  PROC DrawPart12()
    MoveL Offs(pOrigin,195.12,-45.16,-0.00),v40,z0,tcp\WObj:=Plywood;
    MoveL Offs(pOrigin,198.74,-44.14,-0.00),v40,z0,tcp\WObj:=Plywood;
    MoveL Offs(pOrigin,202.88,-41.55,-0.00),v40,z0,tcp\WObj:=Plywood;
    MoveL Offs(pOrigin,205.61,-38.96,-0.00),v40,z0,tcp\WObj:=Plywood;
    MoveL Offs(pOrigin,203.94,-41.12,-0.00),v40,z0,tcp\WObj:=Plywood;
    MoveL Offs(pOrigin,201.82,-42.93,-0.00),v40,z0,tcp\WObj:=Plywood;
    MoveL Offs(pOrigin,198.52,-44.77,-0.00),v40,z0,tcp\WObj:=Plywood;
    MoveL Offs(pOrigin,195.87,-45.59,-0.00),v40,z0,tcp\WObj:=Plywood;
    MoveL Offs(pOrigin,191.41,-45.80,-0.00),v40,z0,tcp\WObj:=Plywood;
    MoveL Offs(pOrigin,188.96,-45.38,-0.00),v40,z0,tcp\WObj:=Plywood;
    MoveL Offs(pOrigin,185.14,-44.24,-0.00),v40,z0,tcp\WObj:=Plywood;
    MoveL Offs(pOrigin,180.14,-41.51,-0.00),v40,z0,tcp\WObj:=Plywood;
    MoveL Offs(pOrigin,177.10,-41.34,-0.00),v40,z0,tcp\WObj:=Plywood;
    MoveL Offs(pOrigin,177.74,-41.62,-0.00),v40,z0,tcp\WObj:=Plywood;
    MoveL Offs(pOrigin,179.93,-44.53,-0.00),v40,z0,tcp\WObj:=Plywood;
    MoveL Offs(pOrigin,183.47,-47.75,-0.00),v40,z0,tcp\WObj:=Plywood;
    MoveL Offs(pOrigin,180.04,-45.06,-0.00),v40,z0,tcp\WObj:=Plywood;
    MoveL Offs(pOrigin,177.74,-41.62,-0.00),v40,fine,tcp\WObj:=Plywood;
    MoveL Offs(pOrigin,177.74,-41.62,-6.00),v60,z5,tcp\WObj:=Plywood;
    MoveL Offs(pOrigin,178.83,-45.34,-6.00),vTravel,z5,tcp\WObj:=Plywood;
    MoveL Offs(pOrigin,178.83,-45.34,-0.00),v60,z0,tcp\WObj:=Plywood;
    MoveL Offs(pOrigin,182.48,-49.09,-0.00),v40,z0,tcp\WObj:=Plywood;
    MoveL Offs(pOrigin,184.50,-50.30,-0.00),v40,z0,tcp\WObj:=Plywood;
    MoveL Offs(pOrigin,186.55,-51.01,-0.00),v40,z0,tcp\WObj:=Plywood;
    MoveL Offs(pOrigin,184.61,-50.51,-0.00),v40,z0,tcp\WObj:=Plywood;
    MoveL Offs(pOrigin,182.16,-49.20,-0.00),v40,z0,tcp\WObj:=Plywood;
    MoveL Offs(pOrigin,180.68,-47.92,-0.00),v40,z0,tcp\WObj:=Plywood;
    MoveL Offs(pOrigin,178.83,-45.34,-0.00),v40,fine,tcp\WObj:=Plywood;
    MoveL Offs(pOrigin,178.83,-45.34,-6.00),v60,z5,tcp\WObj:=Plywood;
    MoveL Offs(pOrigin,183.61,-42.29,-6.00),vTravel,z5,tcp\WObj:=Plywood;
    MoveL Offs(pOrigin,183.61,-42.29,-0.00),v60,z0,tcp\WObj:=Plywood;
    MoveL Offs(pOrigin,187.58,-42.61,-0.00),v40,z0,tcp\WObj:=Plywood;
    MoveL Offs(pOrigin,192.82,-41.76,-0.00),v40,z0,tcp\WObj:=Plywood;
    MoveL Offs(pOrigin,188.32,-42.83,-0.00),v40,z0,tcp\WObj:=Plywood;
    MoveL Offs(pOrigin,185.24,-42.72,-0.00),v40,z0,tcp\WObj:=Plywood;
    MoveL Offs(pOrigin,183.61,-42.29,-0.00),v40,fine,tcp\WObj:=Plywood;
    MoveL Offs(pOrigin,183.61,-42.29,-6.00),v60,z5,tcp\WObj:=Plywood;
    MoveL Offs(pOrigin,189.56,-46.22,-6.00),vTravel,z5,tcp\WObj:=Plywood;
    MoveL Offs(pOrigin,189.56,-46.22,-0.00),v60,z0,tcp\WObj:=Plywood;
    MoveL Offs(pOrigin,194.06,-47.29,-0.00),v40,z0,tcp\WObj:=Plywood;
    MoveL Offs(pOrigin,198.14,-47.08,-0.00),v40,z0,tcp\WObj:=Plywood;
    MoveL Offs(pOrigin,196.40,-47.50,-0.00),v40,z0,tcp\WObj:=Plywood;
    MoveL Offs(pOrigin,193.64,-47.50,-0.00),v40,z0,tcp\WObj:=Plywood;
    MoveL Offs(pOrigin,189.56,-46.22,-0.00),v40,fine,tcp\WObj:=Plywood;
    MoveL Offs(pOrigin,189.56,-46.22,-6.00),v60,z5,tcp\WObj:=Plywood;
    MoveL Offs(pOrigin,191.94,-54.30,-6.00),vTravel,z5,tcp\WObj:=Plywood;
    MoveL Offs(pOrigin,191.94,-54.30,-0.00),v60,z0,tcp\WObj:=Plywood;
    MoveL Offs(pOrigin,195.87,-53.17,-0.00),v40,z0,tcp\WObj:=Plywood;
    MoveL Offs(pOrigin,199.06,-51.68,-0.00),v40,z0,tcp\WObj:=Plywood;
    MoveL Offs(pOrigin,201.85,-49.70,-0.00),v40,z0,tcp\WObj:=Plywood;
    MoveL Offs(pOrigin,199.38,-51.79,-0.00),v40,z0,tcp\WObj:=Plywood;
    MoveL Offs(pOrigin,195.76,-53.59,-0.00),v40,z0,tcp\WObj:=Plywood;
    MoveL Offs(pOrigin,192.26,-54.62,-0.00),v40,z0,tcp\WObj:=Plywood;
    MoveL Offs(pOrigin,188.11,-55.15,-0.00),v40,z0,tcp\WObj:=Plywood;
    MoveL Offs(pOrigin,185.35,-54.94,-0.00),v40,z0,tcp\WObj:=Plywood;
    MoveL Offs(pOrigin,182.91,-54.23,-0.00),v40,z0,tcp\WObj:=Plywood;
    MoveL Offs(pOrigin,180.78,-52.71,-0.00),v40,z0,tcp\WObj:=Plywood;
    MoveL Offs(pOrigin,179.75,-51.01,-0.00),v40,z0,tcp\WObj:=Plywood;
    MoveL Offs(pOrigin,181.21,-52.81,-0.00),v40,z0,tcp\WObj:=Plywood;
    MoveL Offs(pOrigin,183.01,-53.91,-0.00),v40,z0,tcp\WObj:=Plywood;
    MoveL Offs(pOrigin,185.56,-54.62,-0.00),v40,z0,tcp\WObj:=Plywood;
    MoveL Offs(pOrigin,188.75,-54.72,-0.00),v40,z0,tcp\WObj:=Plywood;
    MoveL Offs(pOrigin,191.94,-54.30,-0.00),v40,fine,tcp\WObj:=Plywood;
    MoveL Offs(pOrigin,191.94,-54.30,-6.00),v60,z5,tcp\WObj:=Plywood;
    MoveL Offs(pOrigin,191.30,-56.64,-6.00),vTravel,z5,tcp\WObj:=Plywood;
    MoveL Offs(pOrigin,191.30,-56.64,-0.00),v60,z0,tcp\WObj:=Plywood;
    MoveL Offs(pOrigin,186.20,-56.96,-0.00),v40,z0,tcp\WObj:=Plywood;
    MoveL Offs(pOrigin,182.91,-56.42,-0.00),v40,z0,tcp\WObj:=Plywood;
    MoveL Offs(pOrigin,179.36,-55.04,-0.00),v40,z0,tcp\WObj:=Plywood;
    MoveL Offs(pOrigin,183.23,-56.32,-0.00),v40,z0,tcp\WObj:=Plywood;
    MoveL Offs(pOrigin,186.94,-56.74,-0.00),v40,z0,tcp\WObj:=Plywood;
    MoveL Offs(pOrigin,190.66,-56.53,-0.00),v40,z0,tcp\WObj:=Plywood;
    MoveL Offs(pOrigin,195.59,-55.36,-0.00),v40,z0,tcp\WObj:=Plywood;
    MoveL Offs(pOrigin,191.30,-56.64,-0.00),v40,fine,tcp\WObj:=Plywood;
    MoveL Offs(pOrigin,191.30,-56.64,-6.00),v60,z5,tcp\WObj:=Plywood;
    MoveL Offs(pOrigin,195.80,-66.84,-6.00),vTravel,z5,tcp\WObj:=Plywood;
    MoveL Offs(pOrigin,195.80,-66.84,-0.00),v60,z0,tcp\WObj:=Plywood;
    MoveL Offs(pOrigin,195.44,-67.69,-0.00),v40,z0,tcp\WObj:=Plywood;
    MoveL Offs(pOrigin,195.23,-71.94,-0.00),v40,z0,tcp\WObj:=Plywood;
    MoveL Offs(pOrigin,194.70,-73.21,-0.00),v40,z0,tcp\WObj:=Plywood;
    MoveL Offs(pOrigin,193.39,-74.70,-0.00),v40,z0,tcp\WObj:=Plywood;
    MoveL Offs(pOrigin,193.43,-77.57,-0.00),v40,z0,tcp\WObj:=Plywood;
    MoveL Offs(pOrigin,191.16,-82.56,-0.00),v40,z0,tcp\WObj:=Plywood;
    MoveL Offs(pOrigin,190.34,-85.22,-0.00),v40,z0,tcp\WObj:=Plywood;
    MoveL Offs(pOrigin,190.88,-87.88,-0.00),v40,z0,tcp\WObj:=Plywood;
    MoveL Offs(pOrigin,189.18,-94.25,-0.00),v40,z0,tcp\WObj:=Plywood;
    MoveL Offs(pOrigin,190.66,-103.81,-0.00),v40,z0,tcp\WObj:=Plywood;
    MoveL Offs(pOrigin,190.88,-111.68,-0.00),v40,z0,tcp\WObj:=Plywood;
    MoveL Offs(pOrigin,190.13,-116.56,-0.00),v40,z0,tcp\WObj:=Plywood;
    MoveL Offs(pOrigin,188.86,-119.68,-0.00),v40,z0,tcp\WObj:=Plywood;
    MoveL Offs(pOrigin,190.80,-116.88,-0.00),v40,z0,tcp\WObj:=Plywood;
    MoveL Offs(pOrigin,192.15,-111.57,-0.00),v40,z0,tcp\WObj:=Plywood;
    MoveL Offs(pOrigin,196.40,-67.47,-0.00),v40,z0,tcp\WObj:=Plywood;
    MoveL Offs(pOrigin,196.19,-66.73,-0.00),v40,z0,tcp\WObj:=Plywood;
    MoveL Offs(pOrigin,195.80,-66.84,-0.00),v40,fine,tcp\WObj:=Plywood;
    MoveL Offs(pOrigin,195.80,-66.84,-6.00),v60,z5,tcp\WObj:=Plywood;
    MoveL Offs(pOrigin,193.35,-71.19,-6.00),vTravel,z5,tcp\WObj:=Plywood;
    MoveL Offs(pOrigin,193.35,-71.19,-0.00),v60,z0,tcp\WObj:=Plywood;
    MoveL Offs(pOrigin,191.19,-71.09,-0.00),v40,z0,tcp\WObj:=Plywood;
    MoveL Offs(pOrigin,188.18,-69.64,-0.00),v40,z0,tcp\WObj:=Plywood;
    MoveL Offs(pOrigin,191.30,-70.88,-0.00),v40,z0,tcp\WObj:=Plywood;
    MoveL Offs(pOrigin,193.35,-71.19,-0.00),v40,fine,tcp\WObj:=Plywood;
    MoveL Offs(pOrigin,193.35,-71.19,-6.00),v60,z5,tcp\WObj:=Plywood;
    MoveL Offs(pOrigin,181.52,-78.17,-6.00),vTravel,z5,tcp\WObj:=Plywood;
    MoveL Offs(pOrigin,181.52,-78.17,-0.00),v60,z0,tcp\WObj:=Plywood;
    MoveL Offs(pOrigin,188.04,-89.11,-0.00),v40,z0,tcp\WObj:=Plywood;
    MoveL Offs(pOrigin,184.68,-84.16,-0.00),v40,z0,tcp\WObj:=Plywood;
    MoveL Offs(pOrigin,181.52,-78.17,-0.00),v40,fine,tcp\WObj:=Plywood;
    MoveL Offs(pOrigin,181.52,-78.17,-6.00),v60,z5,tcp\WObj:=Plywood;
    MoveL Offs(pOrigin,172.25,-67.05,-6.00),vTravel,z5,tcp\WObj:=Plywood;
    MoveL Offs(pOrigin,172.25,-67.05,-0.00),v60,z0,tcp\WObj:=Plywood;
    MoveL Offs(pOrigin,172.49,-63.33,-0.00),v40,z0,tcp\WObj:=Plywood;
    MoveL Offs(pOrigin,172.18,-61.88,-0.00),v40,z0,tcp\WObj:=Plywood;
    MoveL Offs(pOrigin,152.73,-56.53,-0.00),v40,z0,tcp\WObj:=Plywood;
    MoveL Offs(pOrigin,148.16,-55.47,-0.00),v40,z0,tcp\WObj:=Plywood;
    MoveL Offs(pOrigin,147.49,-55.79,-0.00),v40,z0,tcp\WObj:=Plywood;
    MoveL Offs(pOrigin,149.01,-60.60,-0.00),v40,z0,tcp\WObj:=Plywood;
    MoveL Offs(pOrigin,172.25,-67.05,-0.00),v40,fine,tcp\WObj:=Plywood;
    MoveL Offs(pOrigin,172.25,-67.05,-6.00),v60,z5,tcp\WObj:=Plywood;
    MoveL Offs(pOrigin,170.83,-65.56,-6.00),vTravel,z5,tcp\WObj:=Plywood;
  ENDPROC

  PROC DrawPart13()
    MoveL Offs(pOrigin,170.83,-65.56,-0.00),v60,z0,tcp\WObj:=Plywood;
    MoveL Offs(pOrigin,151.00,-60.14,-0.00),v40,z0,tcp\WObj:=Plywood;
    MoveL Offs(pOrigin,170.83,-65.56,-0.00),v40,fine,tcp\WObj:=Plywood;
    MoveL Offs(pOrigin,170.83,-65.56,-6.00),v60,z5,tcp\WObj:=Plywood;
    MoveL Offs(pOrigin,155.00,-73.39,-6.00),vTravel,z5,tcp\WObj:=Plywood;
    MoveL Offs(pOrigin,155.00,-73.39,-0.00),v60,z0,tcp\WObj:=Plywood;
    MoveL Offs(pOrigin,158.43,-79.38,-0.00),v40,z0,tcp\WObj:=Plywood;
    MoveL Offs(pOrigin,162.08,-84.58,-0.00),v40,z0,tcp\WObj:=Plywood;
    MoveL Offs(pOrigin,165.48,-88.62,-0.00),v40,z0,tcp\WObj:=Plywood;
    MoveL Offs(pOrigin,170.09,-92.90,-0.00),v40,z0,tcp\WObj:=Plywood;
    MoveL Offs(pOrigin,167.07,-90.53,-0.00),v40,z0,tcp\WObj:=Plywood;
    MoveL Offs(pOrigin,161.76,-84.69,-0.00),v40,z0,tcp\WObj:=Plywood;
    MoveL Offs(pOrigin,157.90,-78.95,-0.00),v40,z0,tcp\WObj:=Plywood;
    MoveL Offs(pOrigin,155.00,-73.39,-0.00),v40,fine,tcp\WObj:=Plywood;
    MoveL Offs(pOrigin,155.00,-73.39,-6.00),v60,z5,tcp\WObj:=Plywood;
    MoveL Offs(pOrigin,152.62,-86.92,-6.00),vTravel,z5,tcp\WObj:=Plywood;
    MoveL Offs(pOrigin,152.62,-86.92,-0.00),v60,z0,tcp\WObj:=Plywood;
    MoveL Offs(pOrigin,153.12,-87.13,-0.00),v40,z0,tcp\WObj:=Plywood;
    MoveL Offs(pOrigin,153.05,-87.52,-0.00),v40,z0,tcp\WObj:=Plywood;
    MoveL Offs(pOrigin,148.27,-89.26,-0.00),v40,z0,tcp\WObj:=Plywood;
    MoveL Offs(pOrigin,147.63,-89.15,-0.00),v40,z0,tcp\WObj:=Plywood;
    MoveL Offs(pOrigin,151.35,-87.31,-0.00),v40,z0,tcp\WObj:=Plywood;
    MoveL Offs(pOrigin,152.62,-86.92,-0.00),v40,z0,tcp\WObj:=Plywood;
    MoveL Offs(pOrigin,152.84,-87.24,-0.00),v40,z0,tcp\WObj:=Plywood;
    MoveL Offs(pOrigin,151.14,-87.63,-0.00),v40,z0,tcp\WObj:=Plywood;
    MoveL Offs(pOrigin,148.55,-88.83,-0.00),v40,z0,tcp\WObj:=Plywood;
    MoveL Offs(pOrigin,151.14,-88.12,-0.00),v40,z0,tcp\WObj:=Plywood;
    MoveL Offs(pOrigin,152.84,-87.24,-0.00),v40,fine,tcp\WObj:=Plywood;
    MoveL Offs(pOrigin,152.84,-87.24,-6.00),v60,z5,tcp\WObj:=Plywood;
    MoveL Offs(pOrigin,159.32,-88.58,-6.00),vTravel,z5,tcp\WObj:=Plywood;
    MoveL Offs(pOrigin,159.32,-88.58,-0.00),v60,z0,tcp\WObj:=Plywood;
    MoveL Offs(pOrigin,160.38,-92.02,-0.00),v40,z0,tcp\WObj:=Plywood;
    MoveL Offs(pOrigin,160.49,-94.89,-0.00),v40,z0,tcp\WObj:=Plywood;
    MoveL Offs(pOrigin,159.50,-98.18,-0.00),v40,z0,tcp\WObj:=Plywood;
    MoveL Offs(pOrigin,157.65,-100.87,-0.00),v40,z0,tcp\WObj:=Plywood;
    MoveL Offs(pOrigin,159.25,-98.18,-0.00),v40,z0,tcp\WObj:=Plywood;
    MoveL Offs(pOrigin,160.17,-95.10,-0.00),v40,z0,tcp\WObj:=Plywood;
    MoveL Offs(pOrigin,160.17,-92.12,-0.00),v40,z0,tcp\WObj:=Plywood;
    MoveL Offs(pOrigin,159.32,-88.58,-0.00),v40,fine,tcp\WObj:=Plywood;
    MoveL Offs(pOrigin,159.32,-88.58,-6.00),v60,z5,tcp\WObj:=Plywood;
    MoveL Offs(pOrigin,156.98,-99.92,-6.00),vTravel,z5,tcp\WObj:=Plywood;
    MoveL Offs(pOrigin,156.98,-99.92,-0.00),v60,z0,tcp\WObj:=Plywood;
    MoveL Offs(pOrigin,150.71,-97.01,-0.00),v40,z0,tcp\WObj:=Plywood;
    MoveL Offs(pOrigin,143.81,-102.01,-0.00),v40,z0,tcp\WObj:=Plywood;
    MoveL Offs(pOrigin,144.87,-109.02,-0.00),v40,z0,tcp\WObj:=Plywood;
    MoveL Offs(pOrigin,144.59,-114.54,-0.00),v40,z0,tcp\WObj:=Plywood;
    MoveL Offs(pOrigin,151.24,-107.43,-0.00),v40,z0,tcp\WObj:=Plywood;
    MoveL Offs(pOrigin,156.98,-99.92,-0.00),v40,fine,tcp\WObj:=Plywood;
    MoveL Offs(pOrigin,156.98,-99.92,-6.00),v60,z5,tcp\WObj:=Plywood;
    MoveL Offs(pOrigin,158.36,-107.04,-6.00),vTravel,z5,tcp\WObj:=Plywood;
    MoveL Offs(pOrigin,158.36,-107.04,-0.00),v60,z0,tcp\WObj:=Plywood;
    MoveL Offs(pOrigin,150.50,-109.30,-0.00),v40,z0,tcp\WObj:=Plywood;
    MoveL Offs(pOrigin,147.10,-112.63,-0.00),v40,z0,tcp\WObj:=Plywood;
    MoveL Offs(pOrigin,144.59,-115.71,-0.00),v40,z0,tcp\WObj:=Plywood;
    MoveL Offs(pOrigin,145.51,-118.47,-0.00),v40,z0,tcp\WObj:=Plywood;
    MoveL Offs(pOrigin,145.97,-121.34,-0.00),v40,z0,tcp\WObj:=Plywood;
    MoveL Offs(pOrigin,147.31,-121.34,-0.00),v40,z0,tcp\WObj:=Plywood;
    MoveL Offs(pOrigin,148.69,-122.19,-0.00),v40,z0,tcp\WObj:=Plywood;
    MoveL Offs(pOrigin,162.61,-121.88,-0.00),v40,z0,tcp\WObj:=Plywood;
    MoveL Offs(pOrigin,175.79,-120.60,-0.00),v40,z0,tcp\WObj:=Plywood;
    MoveL Offs(pOrigin,181.21,-119.54,-0.00),v40,z0,tcp\WObj:=Plywood;
    MoveL Offs(pOrigin,183.23,-118.72,-0.00),v40,z0,tcp\WObj:=Plywood;
    MoveL Offs(pOrigin,184.50,-117.84,-0.00),v40,z0,tcp\WObj:=Plywood;
    MoveL Offs(pOrigin,186.02,-116.03,-0.00),v40,z0,tcp\WObj:=Plywood;
    MoveL Offs(pOrigin,187.26,-112.95,-0.00),v40,z0,tcp\WObj:=Plywood;
    MoveL Offs(pOrigin,187.79,-110.08,-0.00),v40,z0,tcp\WObj:=Plywood;
    MoveL Offs(pOrigin,187.79,-105.62,-0.00),v40,z0,tcp\WObj:=Plywood;
    MoveL Offs(pOrigin,186.27,-97.97,-0.00),v40,z0,tcp\WObj:=Plywood;
    MoveL Offs(pOrigin,185.77,-97.76,-0.00),v40,z0,tcp\WObj:=Plywood;
    MoveL Offs(pOrigin,171.64,-101.79,-0.00),v40,z0,tcp\WObj:=Plywood;
    MoveL Offs(pOrigin,158.36,-107.04,-0.00),v40,fine,tcp\WObj:=Plywood;
    MoveL Offs(pOrigin,158.36,-107.04,-6.00),v60,z5,tcp\WObj:=Plywood;
    MoveL Offs(pOrigin,156.02,-122.62,-6.00),vTravel,z5,tcp\WObj:=Plywood;
    MoveL Offs(pOrigin,156.02,-122.62,-0.00),v60,z0,tcp\WObj:=Plywood;
    MoveL Offs(pOrigin,149.01,-122.44,-0.00),v40,z0,tcp\WObj:=Plywood;
    MoveL Offs(pOrigin,149.54,-124.96,-0.00),v40,z0,tcp\WObj:=Plywood;
    MoveL Offs(pOrigin,158.26,-125.06,-0.00),v40,z0,tcp\WObj:=Plywood;
    MoveL Offs(pOrigin,172.28,-124.21,-0.00),v40,z0,tcp\WObj:=Plywood;
    MoveL Offs(pOrigin,181.95,-122.94,-0.00),v40,z0,tcp\WObj:=Plywood;
    MoveL Offs(pOrigin,185.03,-122.12,-0.00),v40,z0,tcp\WObj:=Plywood;
    MoveL Offs(pOrigin,186.94,-121.24,-0.00),v40,z0,tcp\WObj:=Plywood;
    MoveL Offs(pOrigin,188.57,-119.22,-0.00),v40,z0,tcp\WObj:=Plywood;
    MoveL Offs(pOrigin,189.32,-117.52,-0.00),v40,z0,tcp\WObj:=Plywood;
    MoveL Offs(pOrigin,190.24,-112.31,-0.00),v40,z0,tcp\WObj:=Plywood;
    MoveL Offs(pOrigin,190.24,-105.83,-0.00),v40,z0,tcp\WObj:=Plywood;
    MoveL Offs(pOrigin,189.07,-95.31,-0.00),v40,z0,tcp\WObj:=Plywood;
    MoveL Offs(pOrigin,188.22,-96.59,-0.00),v40,z0,tcp\WObj:=Plywood;
    MoveL Offs(pOrigin,186.84,-97.76,-0.00),v40,z0,tcp\WObj:=Plywood;
    MoveL Offs(pOrigin,188.64,-106.89,-0.00),v40,z0,tcp\WObj:=Plywood;
    MoveL Offs(pOrigin,188.86,-109.97,-0.00),v40,z0,tcp\WObj:=Plywood;
    MoveL Offs(pOrigin,188.64,-114.86,-0.00),v40,z0,tcp\WObj:=Plywood;
    MoveL Offs(pOrigin,187.51,-118.69,-0.00),v40,z0,tcp\WObj:=Plywood;
    MoveL Offs(pOrigin,185.67,-120.81,-0.00),v40,z0,tcp\WObj:=Plywood;
    MoveL Offs(pOrigin,182.59,-122.09,-0.00),v40,z0,tcp\WObj:=Plywood;
    MoveL Offs(pOrigin,179.15,-122.26,-0.00),v40,z0,tcp\WObj:=Plywood;
    MoveL Offs(pOrigin,183.86,-121.06,-0.00),v40,z0,tcp\WObj:=Plywood;
    MoveL Offs(pOrigin,185.24,-120.28,-0.00),v40,z0,tcp\WObj:=Plywood;
    MoveL Offs(pOrigin,186.41,-119.11,-0.00),v40,z0,tcp\WObj:=Plywood;
    MoveL Offs(pOrigin,187.30,-117.52,-0.00),v40,z0,tcp\WObj:=Plywood;
    MoveL Offs(pOrigin,188.01,-114.86,-0.00),v40,z0,tcp\WObj:=Plywood;
    MoveL Offs(pOrigin,188.22,-112.84,-0.00),v40,z0,tcp\WObj:=Plywood;
    MoveL Offs(pOrigin,188.01,-109.41,-0.00),v40,z0,tcp\WObj:=Plywood;
    MoveL Offs(pOrigin,187.48,-112.84,-0.00),v40,z0,tcp\WObj:=Plywood;
    MoveL Offs(pOrigin,186.13,-116.24,-0.00),v40,z0,tcp\WObj:=Plywood;
    MoveL Offs(pOrigin,184.39,-118.26,-0.00),v40,z0,tcp\WObj:=Plywood;
    MoveL Offs(pOrigin,182.38,-119.47,-0.00),v40,z0,tcp\WObj:=Plywood;
    MoveL Offs(pOrigin,177.81,-120.71,-0.00),v40,z0,tcp\WObj:=Plywood;
    MoveL Offs(pOrigin,168.67,-121.88,-0.00),v40,z0,tcp\WObj:=Plywood;
    MoveL Offs(pOrigin,156.02,-122.62,-0.00),v40,fine,tcp\WObj:=Plywood;
    MoveL Offs(pOrigin,156.02,-122.62,-6.00),v60,z5,tcp\WObj:=Plywood;
    MoveL Offs(pOrigin,148.41,-123.04,-6.00),vTravel,z5,tcp\WObj:=Plywood;
    MoveL Offs(pOrigin,148.41,-123.04,-0.00),v60,z0,tcp\WObj:=Plywood;
    MoveL Offs(pOrigin,147.52,-122.02,-0.00),v40,z0,tcp\WObj:=Plywood;
    MoveL Offs(pOrigin,146.78,-121.88,-0.00),v40,z0,tcp\WObj:=Plywood;
    MoveL Offs(pOrigin,146.14,-122.19,-0.00),v40,z0,tcp\WObj:=Plywood;
    MoveL Offs(pOrigin,145.29,-126.27,-0.00),v40,z0,tcp\WObj:=Plywood;
    MoveL Offs(pOrigin,145.51,-122.72,-0.00),v40,z0,tcp\WObj:=Plywood;
    MoveL Offs(pOrigin,144.76,-118.05,-0.00),v40,z0,tcp\WObj:=Plywood;
    MoveL Offs(pOrigin,143.31,-114.76,-0.00),v40,z0,tcp\WObj:=Plywood;
    MoveL Offs(pOrigin,140.23,-110.15,-0.00),v40,z0,tcp\WObj:=Plywood;
  ENDPROC

  PROC DrawPart14()
    MoveL Offs(pOrigin,143.59,-114.37,-0.00),v40,z0,tcp\WObj:=Plywood;
    MoveL Offs(pOrigin,142.35,-110.40,-0.00),v40,z0,tcp\WObj:=Plywood;
    MoveL Offs(pOrigin,141.08,-107.85,-0.00),v40,z0,tcp\WObj:=Plywood;
    MoveL Offs(pOrigin,139.56,-105.83,-0.00),v40,z0,tcp\WObj:=Plywood;
    MoveL Offs(pOrigin,134.85,-102.15,-0.00),v40,z0,tcp\WObj:=Plywood;
    MoveL Offs(pOrigin,137.75,-103.81,-0.00),v40,z0,tcp\WObj:=Plywood;
    MoveL Offs(pOrigin,139.84,-105.51,-0.00),v40,z0,tcp\WObj:=Plywood;
    MoveL Offs(pOrigin,137.96,-102.22,-0.00),v40,z0,tcp\WObj:=Plywood;
    MoveL Offs(pOrigin,135.52,-100.27,-0.00),v40,z0,tcp\WObj:=Plywood;
    MoveL Offs(pOrigin,132.86,-98.89,-0.00),v40,z0,tcp\WObj:=Plywood;
    MoveL Offs(pOrigin,129.89,-98.07,-0.00),v40,z0,tcp\WObj:=Plywood;
    MoveL Offs(pOrigin,126.66,-98.39,-0.00),v40,z0,tcp\WObj:=Plywood;
    MoveL Offs(pOrigin,128.93,-97.86,-0.00),v40,z0,tcp\WObj:=Plywood;
    MoveL Offs(pOrigin,131.38,-98.18,-0.00),v40,z0,tcp\WObj:=Plywood;
    MoveL Offs(pOrigin,133.39,-98.89,-0.00),v40,z0,tcp\WObj:=Plywood;
    MoveL Offs(pOrigin,137.40,-101.16,-0.00),v40,z0,tcp\WObj:=Plywood;
    MoveL Offs(pOrigin,135.52,-98.18,-0.00),v40,z0,tcp\WObj:=Plywood;
    MoveL Offs(pOrigin,134.46,-97.12,-0.00),v40,z0,tcp\WObj:=Plywood;
    MoveL Offs(pOrigin,130.81,-95.21,-0.00),v40,z0,tcp\WObj:=Plywood;
    MoveL Offs(pOrigin,134.53,-96.69,-0.00),v40,z0,tcp\WObj:=Plywood;
    MoveL Offs(pOrigin,130.84,-91.70,-0.00),v40,z0,tcp\WObj:=Plywood;
    MoveL Offs(pOrigin,129.04,-86.92,-0.00),v40,z0,tcp\WObj:=Plywood;
    MoveL Offs(pOrigin,126.49,-84.72,-0.00),v40,z0,tcp\WObj:=Plywood;
    MoveL Offs(pOrigin,122.73,-87.98,-0.00),v40,z0,tcp\WObj:=Plywood;
    MoveL Offs(pOrigin,121.00,-92.76,-0.00),v40,z0,tcp\WObj:=Plywood;
    MoveL Offs(pOrigin,122.59,-92.27,-0.00),v40,z0,tcp\WObj:=Plywood;
    MoveL Offs(pOrigin,120.64,-93.40,-0.00),v40,z0,tcp\WObj:=Plywood;
    MoveL Offs(pOrigin,119.40,-95.63,-0.00),v40,z0,tcp\WObj:=Plywood;
    MoveL Offs(pOrigin,123.44,-94.46,-0.00),v40,z0,tcp\WObj:=Plywood;
    MoveL Offs(pOrigin,121.18,-95.17,-0.00),v40,z0,tcp\WObj:=Plywood;
    MoveL Offs(pOrigin,118.62,-96.69,-0.00),v40,z0,tcp\WObj:=Plywood;
    MoveL Offs(pOrigin,116.22,-100.09,-0.00),v40,z0,tcp\WObj:=Plywood;
    MoveL Offs(pOrigin,119.16,-98.57,-0.00),v40,z0,tcp\WObj:=Plywood;
    MoveL Offs(pOrigin,122.27,-97.97,-0.00),v40,z0,tcp\WObj:=Plywood;
    MoveL Offs(pOrigin,119.16,-98.78,-0.00),v40,z0,tcp\WObj:=Plywood;
    MoveL Offs(pOrigin,116.29,-100.62,-0.00),v40,z0,tcp\WObj:=Plywood;
    MoveL Offs(pOrigin,114.80,-102.32,-0.00),v40,z0,tcp\WObj:=Plywood;
    MoveL Offs(pOrigin,113.95,-103.99,-0.00),v40,z0,tcp\WObj:=Plywood;
    MoveL Offs(pOrigin,116.93,-102.29,-0.00),v40,z0,tcp\WObj:=Plywood;
    MoveL Offs(pOrigin,119.62,-101.37,-0.00),v40,z0,tcp\WObj:=Plywood;
    MoveL Offs(pOrigin,116.50,-102.82,-0.00),v40,z0,tcp\WObj:=Plywood;
    MoveL Offs(pOrigin,113.84,-104.66,-0.00),v40,z0,tcp\WObj:=Plywood;
    MoveL Offs(pOrigin,110.37,-108.28,-0.00),v40,z0,tcp\WObj:=Plywood;
    MoveL Offs(pOrigin,113.24,-107.11,-0.00),v40,z0,tcp\WObj:=Plywood;
    MoveL Offs(pOrigin,110.02,-108.91,-0.00),v40,z0,tcp\WObj:=Plywood;
    MoveL Offs(pOrigin,107.04,-111.68,-0.00),v40,z0,tcp\WObj:=Plywood;
    MoveL Offs(pOrigin,104.99,-115.18,-0.00),v40,z0,tcp\WObj:=Plywood;
    MoveL Offs(pOrigin,103.54,-121.06,-0.00),v40,z0,tcp\WObj:=Plywood;
    MoveL Offs(pOrigin,103.82,-116.67,-0.00),v40,z0,tcp\WObj:=Plywood;
    MoveL Offs(pOrigin,103.01,-116.70,-0.00),v40,z0,tcp\WObj:=Plywood;
    MoveL Offs(pOrigin,102.19,-117.52,-0.00),v40,z0,tcp\WObj:=Plywood;
    MoveL Offs(pOrigin,100.92,-123.68,-0.00),v40,z0,tcp\WObj:=Plywood;
    MoveL Offs(pOrigin,98.12,-129.42,-0.00),v40,z0,tcp\WObj:=Plywood;
    MoveL Offs(pOrigin,98.01,-130.91,-0.00),v40,z0,tcp\WObj:=Plywood;
    MoveL Offs(pOrigin,98.40,-132.93,-0.00),v40,z0,tcp\WObj:=Plywood;
    MoveL Offs(pOrigin,98.97,-133.77,-0.00),v40,z0,tcp\WObj:=Plywood;
    MoveL Offs(pOrigin,100.14,-134.20,-0.00),v40,z0,tcp\WObj:=Plywood;
    MoveL Offs(pOrigin,101.20,-133.56,-0.00),v40,z0,tcp\WObj:=Plywood;
    MoveL Offs(pOrigin,101.70,-132.61,-0.00),v40,z0,tcp\WObj:=Plywood;
    MoveL Offs(pOrigin,101.62,-132.04,-0.00),v40,z0,tcp\WObj:=Plywood;
    MoveL Offs(pOrigin,100.03,-132.71,-0.00),v40,z0,tcp\WObj:=Plywood;
    MoveL Offs(pOrigin,99.39,-132.61,-0.00),v40,z0,tcp\WObj:=Plywood;
    MoveL Offs(pOrigin,98.97,-130.16,-0.00),v40,z0,tcp\WObj:=Plywood;
    MoveL Offs(pOrigin,99.96,-127.68,-0.00),v40,z0,tcp\WObj:=Plywood;
    MoveL Offs(pOrigin,99.18,-129.84,-0.00),v40,z0,tcp\WObj:=Plywood;
    MoveL Offs(pOrigin,99.46,-131.86,-0.00),v40,z0,tcp\WObj:=Plywood;
    MoveL Offs(pOrigin,100.35,-132.29,-0.00),v40,z0,tcp\WObj:=Plywood;
    MoveL Offs(pOrigin,101.59,-131.23,-0.00),v40,z0,tcp\WObj:=Plywood;
    MoveL Offs(pOrigin,102.72,-127.08,-0.00),v40,z0,tcp\WObj:=Plywood;
    MoveL Offs(pOrigin,103.22,-126.55,-0.00),v40,z0,tcp\WObj:=Plywood;
    MoveL Offs(pOrigin,103.18,-124.00,-0.00),v40,z0,tcp\WObj:=Plywood;
    MoveL Offs(pOrigin,102.58,-124.85,-0.00),v40,z0,tcp\WObj:=Plywood;
    MoveL Offs(pOrigin,102.55,-126.48,-0.00),v40,z0,tcp\WObj:=Plywood;
    MoveL Offs(pOrigin,102.37,-124.64,-0.00),v40,z0,tcp\WObj:=Plywood;
    MoveL Offs(pOrigin,103.40,-122.55,-0.00),v40,z0,tcp\WObj:=Plywood;
    MoveL Offs(pOrigin,103.54,-131.90,-0.00),v40,z0,tcp\WObj:=Plywood;
    MoveL Offs(pOrigin,104.64,-128.99,-0.00),v40,z0,tcp\WObj:=Plywood;
    MoveL Offs(pOrigin,105.24,-128.04,-0.00),v40,z0,tcp\WObj:=Plywood;
    MoveL Offs(pOrigin,106.09,-127.47,-0.00),v40,z0,tcp\WObj:=Plywood;
    MoveL Offs(pOrigin,109.38,-127.08,-0.00),v40,z0,tcp\WObj:=Plywood;
    MoveL Offs(pOrigin,114.06,-127.61,-0.00),v40,z0,tcp\WObj:=Plywood;
    MoveL Offs(pOrigin,116.18,-128.21,-0.00),v40,z0,tcp\WObj:=Plywood;
    MoveL Offs(pOrigin,117.56,-129.21,-0.00),v40,z0,tcp\WObj:=Plywood;
    MoveL Offs(pOrigin,118.84,-131.01,-0.00),v40,z0,tcp\WObj:=Plywood;
    MoveL Offs(pOrigin,119.16,-134.41,-0.00),v40,z0,tcp\WObj:=Plywood;
    MoveL Offs(pOrigin,118.73,-134.09,-0.00),v40,z0,tcp\WObj:=Plywood;
    MoveL Offs(pOrigin,118.80,-134.73,-0.00),v40,z0,tcp\WObj:=Plywood;
    MoveL Offs(pOrigin,119.37,-135.19,-0.00),v40,z0,tcp\WObj:=Plywood;
    MoveL Offs(pOrigin,121.18,-135.58,-0.00),v40,z0,tcp\WObj:=Plywood;
    MoveL Offs(pOrigin,122.45,-135.26,-0.00),v40,z0,tcp\WObj:=Plywood;
    MoveL Offs(pOrigin,123.16,-132.71,-0.00),v40,z0,tcp\WObj:=Plywood;
    MoveL Offs(pOrigin,125.85,-129.81,-0.00),v40,z0,tcp\WObj:=Plywood;
    MoveL Offs(pOrigin,127.34,-129.42,-0.00),v40,z0,tcp\WObj:=Plywood;
    MoveL Offs(pOrigin,132.01,-129.63,-0.00),v40,z0,tcp\WObj:=Plywood;
    MoveL Offs(pOrigin,135.41,-130.38,-0.00),v40,z0,tcp\WObj:=Plywood;
    MoveL Offs(pOrigin,137.54,-131.44,-0.00),v40,z0,tcp\WObj:=Plywood;
    MoveL Offs(pOrigin,138.28,-133.46,-0.00),v40,z0,tcp\WObj:=Plywood;
    MoveL Offs(pOrigin,138.53,-137.28,-0.00),v40,z0,tcp\WObj:=Plywood;
    MoveL Offs(pOrigin,140.73,-137.88,-0.00),v40,z0,tcp\WObj:=Plywood;
    MoveL Offs(pOrigin,141.57,-137.88,-0.00),v40,z0,tcp\WObj:=Plywood;
    MoveL Offs(pOrigin,141.96,-137.39,-0.00),v40,z0,tcp\WObj:=Plywood;
    MoveL Offs(pOrigin,143.35,-132.61,-0.00),v40,z0,tcp\WObj:=Plywood;
    MoveL Offs(pOrigin,143.88,-131.76,-0.00),v40,z0,tcp\WObj:=Plywood;
    MoveL Offs(pOrigin,144.55,-132.89,-0.00),v40,z0,tcp\WObj:=Plywood;
    MoveL Offs(pOrigin,145.86,-130.91,-0.00),v40,z0,tcp\WObj:=Plywood;
    MoveL Offs(pOrigin,146.04,-129.74,-0.00),v40,z0,tcp\WObj:=Plywood;
    MoveL Offs(pOrigin,145.19,-127.61,-0.00),v40,z0,tcp\WObj:=Plywood;
    MoveL Offs(pOrigin,145.40,-127.15,-0.00),v40,z0,tcp\WObj:=Plywood;
    MoveL Offs(pOrigin,147.14,-129.21,-0.00),v40,z0,tcp\WObj:=Plywood;
    MoveL Offs(pOrigin,147.42,-130.62,-0.00),v40,z0,tcp\WObj:=Plywood;
    MoveL Offs(pOrigin,146.78,-129.31,-0.00),v40,z0,tcp\WObj:=Plywood;
    MoveL Offs(pOrigin,146.18,-128.89,-0.00),v40,z0,tcp\WObj:=Plywood;
    MoveL Offs(pOrigin,146.46,-130.27,-0.00),v40,z0,tcp\WObj:=Plywood;
    MoveL Offs(pOrigin,145.08,-132.71,-0.00),v40,z0,tcp\WObj:=Plywood;
    MoveL Offs(pOrigin,145.19,-133.14,-0.00),v40,z0,tcp\WObj:=Plywood;
    MoveL Offs(pOrigin,145.86,-133.17,-0.00),v40,z0,tcp\WObj:=Plywood;
    MoveL Offs(pOrigin,145.19,-133.56,-0.00),v40,z0,tcp\WObj:=Plywood;
    MoveL Offs(pOrigin,145.08,-133.99,-0.00),v40,z0,tcp\WObj:=Plywood;
    MoveL Offs(pOrigin,146.36,-136.64,-0.00),v40,z0,tcp\WObj:=Plywood;
    MoveL Offs(pOrigin,147.52,-137.74,-0.00),v40,z0,tcp\WObj:=Plywood;
  ENDPROC

  PROC DrawPart15()
    MoveL Offs(pOrigin,148.27,-137.92,-0.00),v40,z0,tcp\WObj:=Plywood;
    MoveL Offs(pOrigin,149.47,-136.64,-0.00),v40,z0,tcp\WObj:=Plywood;
    MoveL Offs(pOrigin,149.86,-133.99,-0.00),v40,z0,tcp\WObj:=Plywood;
    MoveL Offs(pOrigin,149.23,-131.90,-0.00),v40,z0,tcp\WObj:=Plywood;
    MoveL Offs(pOrigin,148.27,-135.19,-0.00),v40,z0,tcp\WObj:=Plywood;
    MoveL Offs(pOrigin,149.01,-131.12,-0.00),v40,z0,tcp\WObj:=Plywood;
    MoveL Offs(pOrigin,148.52,-128.99,-0.00),v40,z0,tcp\WObj:=Plywood;
    MoveL Offs(pOrigin,147.67,-127.36,-0.00),v40,z0,tcp\WObj:=Plywood;
    MoveL Offs(pOrigin,148.73,-128.99,-0.00),v40,z0,tcp\WObj:=Plywood;
    MoveL Offs(pOrigin,149.97,-133.88,-0.00),v40,z0,tcp\WObj:=Plywood;
    MoveL Offs(pOrigin,150.07,-135.05,-0.00),v40,z0,tcp\WObj:=Plywood;
    MoveL Offs(pOrigin,149.69,-136.75,-0.00),v40,z0,tcp\WObj:=Plywood;
    MoveL Offs(pOrigin,148.59,-138.17,-0.00),v40,z0,tcp\WObj:=Plywood;
    MoveL Offs(pOrigin,147.95,-138.24,-0.00),v40,z0,tcp\WObj:=Plywood;
    MoveL Offs(pOrigin,146.89,-137.71,-0.00),v40,z0,tcp\WObj:=Plywood;
    MoveL Offs(pOrigin,145.79,-136.22,-0.00),v40,z0,tcp\WObj:=Plywood;
    MoveL Offs(pOrigin,144.66,-132.89,-0.00),v40,z0,tcp\WObj:=Plywood;
    MoveL Offs(pOrigin,144.44,-133.24,-0.00),v40,z0,tcp\WObj:=Plywood;
    MoveL Offs(pOrigin,144.69,-135.16,-0.00),v40,z0,tcp\WObj:=Plywood;
    MoveL Offs(pOrigin,145.05,-135.44,-0.00),v40,z0,tcp\WObj:=Plywood;
    MoveL Offs(pOrigin,144.51,-135.79,-0.00),v40,z0,tcp\WObj:=Plywood;
    MoveL Offs(pOrigin,145.08,-136.11,-0.00),v40,z0,tcp\WObj:=Plywood;
    MoveL Offs(pOrigin,144.27,-136.86,-0.00),v40,z0,tcp\WObj:=Plywood;
    MoveL Offs(pOrigin,145.22,-137.46,-0.00),v40,z0,tcp\WObj:=Plywood;
    MoveL Offs(pOrigin,145.40,-138.20,-0.00),v40,z0,tcp\WObj:=Plywood;
    MoveL Offs(pOrigin,147.10,-139.44,-0.00),v40,z0,tcp\WObj:=Plywood;
    MoveL Offs(pOrigin,148.91,-139.44,-0.00),v40,z0,tcp\WObj:=Plywood;
    MoveL Offs(pOrigin,149.76,-138.66,-0.00),v40,z0,tcp\WObj:=Plywood;
    MoveL Offs(pOrigin,150.54,-137.18,-0.00),v40,z0,tcp\WObj:=Plywood;
    MoveL Offs(pOrigin,151.03,-135.48,-0.00),v40,z0,tcp\WObj:=Plywood;
    MoveL Offs(pOrigin,151.03,-133.99,-0.00),v40,z0,tcp\WObj:=Plywood;
    MoveL Offs(pOrigin,148.41,-123.04,-0.00),v40,fine,tcp\WObj:=Plywood;
    MoveL Offs(pOrigin,148.41,-123.04,-6.00),v60,z5,tcp\WObj:=Plywood;
    MoveL Offs(pOrigin,145.36,-132.89,-6.00),vTravel,z5,tcp\WObj:=Plywood;
    MoveL Offs(pOrigin,145.36,-132.89,-0.00),v60,z0,tcp\WObj:=Plywood;
    MoveL Offs(pOrigin,146.39,-131.61,-0.00),v40,z0,tcp\WObj:=Plywood;
    MoveL Offs(pOrigin,145.36,-132.89,-0.00),v40,fine,tcp\WObj:=Plywood;
    MoveL Offs(pOrigin,145.36,-132.89,-6.00),v60,z5,tcp\WObj:=Plywood;
    MoveL Offs(pOrigin,143.17,-136.43,-6.00),vTravel,z5,tcp\WObj:=Plywood;
    MoveL Offs(pOrigin,143.17,-136.43,-0.00),v60,z0,tcp\WObj:=Plywood;
    MoveL Offs(pOrigin,143.59,-136.22,-0.00),v40,z0,tcp\WObj:=Plywood;
    MoveL Offs(pOrigin,143.17,-136.43,-0.00),v40,z0,tcp\WObj:=Plywood;
    MoveL Offs(pOrigin,143.38,-136.79,-0.00),v40,z0,tcp\WObj:=Plywood;
    MoveL Offs(pOrigin,142.99,-137.28,-0.00),v40,z0,tcp\WObj:=Plywood;
    MoveL Offs(pOrigin,143.66,-136.86,-0.00),v40,z0,tcp\WObj:=Plywood;
    MoveL Offs(pOrigin,143.38,-136.79,-0.00),v40,fine,tcp\WObj:=Plywood;
    MoveL Offs(pOrigin,143.38,-136.79,-6.00),v60,z5,tcp\WObj:=Plywood;
    MoveL Offs(pOrigin,143.95,-138.66,-6.00),vTravel,z5,tcp\WObj:=Plywood;
    MoveL Offs(pOrigin,143.95,-138.66,-0.00),v60,z0,tcp\WObj:=Plywood;
    MoveL Offs(pOrigin,140.09,-137.92,-0.00),v40,z0,tcp\WObj:=Plywood;
    MoveL Offs(pOrigin,139.73,-138.77,-0.00),v40,z0,tcp\WObj:=Plywood;
    MoveL Offs(pOrigin,142.96,-138.98,-0.00),v40,z0,tcp\WObj:=Plywood;
    MoveL Offs(pOrigin,143.95,-138.66,-0.00),v40,z0,tcp\WObj:=Plywood;
    MoveL Offs(pOrigin,144.23,-139.19,-0.00),v40,z0,tcp\WObj:=Plywood;
    MoveL Offs(pOrigin,142.32,-139.83,-0.00),v40,z0,tcp\WObj:=Plywood;
    MoveL Offs(pOrigin,141.57,-141.00,-0.00),v40,z0,tcp\WObj:=Plywood;
    MoveL Offs(pOrigin,143.81,-139.73,-0.00),v40,z0,tcp\WObj:=Plywood;
    MoveL Offs(pOrigin,146.39,-139.83,-0.00),v40,z0,tcp\WObj:=Plywood;
    MoveL Offs(pOrigin,144.23,-139.19,-0.00),v40,z0,tcp\WObj:=Plywood;
    MoveL Offs(pOrigin,144.83,-139.94,-0.00),v40,z0,tcp\WObj:=Plywood;
    MoveL Offs(pOrigin,145.86,-140.04,-0.00),v40,z0,tcp\WObj:=Plywood;
    MoveL Offs(pOrigin,144.83,-139.94,-0.00),v40,z0,tcp\WObj:=Plywood;
    MoveL Offs(pOrigin,144.98,-140.61,-0.00),v40,z0,tcp\WObj:=Plywood;
    MoveL Offs(pOrigin,142.96,-141.11,-0.00),v40,z0,tcp\WObj:=Plywood;
    MoveL Offs(pOrigin,139.49,-145.92,-0.00),v40,z0,tcp\WObj:=Plywood;
    MoveL Offs(pOrigin,140.69,-143.66,-0.00),v40,z0,tcp\WObj:=Plywood;
    MoveL Offs(pOrigin,139.38,-144.97,-0.00),v40,z0,tcp\WObj:=Plywood;
    MoveL Offs(pOrigin,140.58,-142.81,-0.00),v40,z0,tcp\WObj:=Plywood;
    MoveL Offs(pOrigin,139.52,-143.83,-0.00),v40,z0,tcp\WObj:=Plywood;
    MoveL Offs(pOrigin,141.15,-139.41,-0.00),v40,z0,tcp\WObj:=Plywood;
    MoveL Offs(pOrigin,140.83,-139.09,-0.00),v40,z0,tcp\WObj:=Plywood;
    MoveL Offs(pOrigin,137.86,-138.98,-0.00),v40,z0,tcp\WObj:=Plywood;
    MoveL Offs(pOrigin,136.48,-139.73,-0.00),v40,z0,tcp\WObj:=Plywood;
    MoveL Offs(pOrigin,131.27,-140.65,-0.00),v40,z0,tcp\WObj:=Plywood;
    MoveL Offs(pOrigin,125.53,-139.65,-0.00),v40,z0,tcp\WObj:=Plywood;
    MoveL Offs(pOrigin,122.88,-137.49,-0.00),v40,z0,tcp\WObj:=Plywood;
    MoveL Offs(pOrigin,121.88,-138.56,-0.00),v40,z0,tcp\WObj:=Plywood;
    MoveL Offs(pOrigin,121.18,-140.72,-0.00),v40,z0,tcp\WObj:=Plywood;
    MoveL Offs(pOrigin,121.67,-138.45,-0.00),v40,z0,tcp\WObj:=Plywood;
    MoveL Offs(pOrigin,122.66,-137.07,-0.00),v40,z0,tcp\WObj:=Plywood;
    MoveL Offs(pOrigin,122.24,-136.43,-0.00),v40,z0,tcp\WObj:=Plywood;
    MoveL Offs(pOrigin,120.86,-136.54,-0.00),v40,z0,tcp\WObj:=Plywood;
    MoveL Offs(pOrigin,118.41,-136.01,-0.00),v40,z0,tcp\WObj:=Plywood;
    MoveL Offs(pOrigin,118.09,-139.55,-0.00),v40,z0,tcp\WObj:=Plywood;
    MoveL Offs(pOrigin,117.88,-137.18,-0.00),v40,z0,tcp\WObj:=Plywood;
    MoveL Offs(pOrigin,117.56,-136.86,-0.00),v40,z0,tcp\WObj:=Plywood;
    MoveL Offs(pOrigin,115.01,-137.74,-0.00),v40,z0,tcp\WObj:=Plywood;
    MoveL Offs(pOrigin,115.69,-137.95,-0.00),v40,z0,tcp\WObj:=Plywood;
    MoveL Offs(pOrigin,115.22,-138.41,-0.00),v40,z0,tcp\WObj:=Plywood;
    MoveL Offs(pOrigin,115.76,-138.27,-0.00),v40,z0,tcp\WObj:=Plywood;
    MoveL Offs(pOrigin,114.06,-138.45,-0.00),v40,z0,tcp\WObj:=Plywood;
    MoveL Offs(pOrigin,108.74,-137.60,-0.00),v40,z0,tcp\WObj:=Plywood;
    MoveL Offs(pOrigin,107.68,-136.82,-0.00),v40,z0,tcp\WObj:=Plywood;
    MoveL Offs(pOrigin,103.43,-135.09,-0.00),v40,z0,tcp\WObj:=Plywood;
    MoveL Offs(pOrigin,102.76,-139.26,-0.00),v40,z0,tcp\WObj:=Plywood;
    MoveL Offs(pOrigin,102.58,-138.66,-0.00),v40,z0,tcp\WObj:=Plywood;
    MoveL Offs(pOrigin,102.37,-138.77,-0.00),v40,z0,tcp\WObj:=Plywood;
    MoveL Offs(pOrigin,102.65,-140.72,-0.00),v40,z0,tcp\WObj:=Plywood;
    MoveL Offs(pOrigin,102.33,-139.94,-0.00),v40,z0,tcp\WObj:=Plywood;
    MoveL Offs(pOrigin,102.05,-140.04,-0.00),v40,z0,tcp\WObj:=Plywood;
    MoveL Offs(pOrigin,102.65,-142.31,-0.00),v40,z0,tcp\WObj:=Plywood;
    MoveL Offs(pOrigin,100.63,-137.07,-0.00),v40,z0,tcp\WObj:=Plywood;
    MoveL Offs(pOrigin,100.28,-136.86,-0.00),v40,z0,tcp\WObj:=Plywood;
    MoveL Offs(pOrigin,100.42,-138.13,-0.00),v40,z0,tcp\WObj:=Plywood;
    MoveL Offs(pOrigin,102.47,-143.66,-0.00),v40,z0,tcp\WObj:=Plywood;
    MoveL Offs(pOrigin,101.77,-142.81,-0.00),v40,z0,tcp\WObj:=Plywood;
    MoveL Offs(pOrigin,103.04,-147.20,-0.00),v40,z0,tcp\WObj:=Plywood;
    MoveL Offs(pOrigin,102.05,-145.46,-0.00),v40,z0,tcp\WObj:=Plywood;
    MoveL Offs(pOrigin,101.84,-145.57,-0.00),v40,z0,tcp\WObj:=Plywood;
    MoveL Offs(pOrigin,103.50,-148.90,-0.00),v40,z0,tcp\WObj:=Plywood;
    MoveL Offs(pOrigin,102.40,-147.80,-0.00),v40,z0,tcp\WObj:=Plywood;
    MoveL Offs(pOrigin,104.21,-150.42,-0.00),v40,z0,tcp\WObj:=Plywood;
    MoveL Offs(pOrigin,101.84,-147.91,-0.00),v40,z0,tcp\WObj:=Plywood;
    MoveL Offs(pOrigin,101.59,-148.01,-0.00),v40,z0,tcp\WObj:=Plywood;
    MoveL Offs(pOrigin,102.69,-149.61,-0.00),v40,z0,tcp\WObj:=Plywood;
    MoveL Offs(pOrigin,104.99,-151.80,-0.00),v40,z0,tcp\WObj:=Plywood;
    MoveL Offs(pOrigin,103.43,-150.92,-0.00),v40,z0,tcp\WObj:=Plywood;
    MoveL Offs(pOrigin,103.54,-151.31,-0.00),v40,z0,tcp\WObj:=Plywood;
    MoveL Offs(pOrigin,105.59,-153.11,-0.00),v40,z0,tcp\WObj:=Plywood;
    MoveL Offs(pOrigin,103.75,-152.37,-0.00),v40,z0,tcp\WObj:=Plywood;
  ENDPROC

  PROC DrawPart16()
    MoveL Offs(pOrigin,103.64,-152.58,-0.00),v40,z0,tcp\WObj:=Plywood;
    MoveL Offs(pOrigin,106.76,-154.25,-0.00),v40,z0,tcp\WObj:=Plywood;
    MoveL Offs(pOrigin,104.07,-153.82,-0.00),v40,z0,tcp\WObj:=Plywood;
    MoveL Offs(pOrigin,107.29,-155.02,-0.00),v40,z0,tcp\WObj:=Plywood;
    MoveL Offs(pOrigin,104.71,-155.13,-0.00),v40,z0,tcp\WObj:=Plywood;
    MoveL Offs(pOrigin,107.82,-155.66,-0.00),v40,z0,tcp\WObj:=Plywood;
    MoveL Offs(pOrigin,105.98,-155.66,-0.00),v40,z0,tcp\WObj:=Plywood;
    MoveL Offs(pOrigin,105.45,-155.88,-0.00),v40,z0,tcp\WObj:=Plywood;
    MoveL Offs(pOrigin,105.56,-156.09,-0.00),v40,z0,tcp\WObj:=Plywood;
    MoveL Offs(pOrigin,107.36,-155.98,-0.00),v40,z0,tcp\WObj:=Plywood;
    MoveL Offs(pOrigin,109.10,-156.30,-0.00),v40,z0,tcp\WObj:=Plywood;
    MoveL Offs(pOrigin,107.26,-156.76,-0.00),v40,z0,tcp\WObj:=Plywood;
    MoveL Offs(pOrigin,107.26,-157.04,-0.00),v40,z0,tcp\WObj:=Plywood;
    MoveL Offs(pOrigin,108.64,-156.73,-0.00),v40,z0,tcp\WObj:=Plywood;
    MoveL Offs(pOrigin,110.27,-156.83,-0.00),v40,z0,tcp\WObj:=Plywood;
    MoveL Offs(pOrigin,109.49,-157.26,-0.00),v40,z0,tcp\WObj:=Plywood;
    MoveL Offs(pOrigin,109.59,-157.47,-0.00),v40,z0,tcp\WObj:=Plywood;
    MoveL Offs(pOrigin,111.40,-157.08,-0.00),v40,z0,tcp\WObj:=Plywood;
    MoveL Offs(pOrigin,110.02,-158.53,-0.00),v40,z0,tcp\WObj:=Plywood;
    MoveL Offs(pOrigin,109.70,-159.35,-0.00),v40,z0,tcp\WObj:=Plywood;
    MoveL Offs(pOrigin,110.97,-158.07,-0.00),v40,z0,tcp\WObj:=Plywood;
    MoveL Offs(pOrigin,112.57,-157.47,-0.00),v40,z0,tcp\WObj:=Plywood;
    MoveL Offs(pOrigin,112.75,-157.79,-0.00),v40,z0,tcp\WObj:=Plywood;
    MoveL Offs(pOrigin,111.82,-159.38,-0.00),v40,z0,tcp\WObj:=Plywood;
    MoveL Offs(pOrigin,112.14,-161.01,-0.00),v40,z0,tcp\WObj:=Plywood;
    MoveL Offs(pOrigin,112.64,-158.74,-0.00),v40,z0,tcp\WObj:=Plywood;
    MoveL Offs(pOrigin,113.31,-157.89,-0.00),v40,z0,tcp\WObj:=Plywood;
    MoveL Offs(pOrigin,114.06,-157.57,-0.00),v40,z0,tcp\WObj:=Plywood;
    MoveL Offs(pOrigin,113.49,-158.43,-0.00),v40,z0,tcp\WObj:=Plywood;
    MoveL Offs(pOrigin,113.31,-159.70,-0.00),v40,z0,tcp\WObj:=Plywood;
    MoveL Offs(pOrigin,114.16,-161.54,-0.00),v40,z0,tcp\WObj:=Plywood;
    MoveL Offs(pOrigin,113.84,-160.34,-0.00),v40,z0,tcp\WObj:=Plywood;
    MoveL Offs(pOrigin,114.13,-158.64,-0.00),v40,z0,tcp\WObj:=Plywood;
    MoveL Offs(pOrigin,114.87,-157.86,-0.00),v40,z0,tcp\WObj:=Plywood;
    MoveL Offs(pOrigin,114.27,-159.49,-0.00),v40,z0,tcp\WObj:=Plywood;
    MoveL Offs(pOrigin,114.48,-160.80,-0.00),v40,z0,tcp\WObj:=Plywood;
    MoveL Offs(pOrigin,114.98,-158.74,-0.00),v40,z0,tcp\WObj:=Plywood;
    MoveL Offs(pOrigin,115.47,-158.14,-0.00),v40,z0,tcp\WObj:=Plywood;
    MoveL Offs(pOrigin,115.12,-159.27,-0.00),v40,z0,tcp\WObj:=Plywood;
    MoveL Offs(pOrigin,115.22,-160.27,-0.00),v40,z0,tcp\WObj:=Plywood;
    MoveL Offs(pOrigin,116.11,-157.82,-0.00),v40,z0,tcp\WObj:=Plywood;
    MoveL Offs(pOrigin,115.65,-159.27,-0.00),v40,z0,tcp\WObj:=Plywood;
    MoveL Offs(pOrigin,115.76,-160.34,-0.00),v40,z0,tcp\WObj:=Plywood;
    MoveL Offs(pOrigin,116.29,-161.51,-0.00),v40,z0,tcp\WObj:=Plywood;
    MoveL Offs(pOrigin,117.46,-162.50,-0.00),v40,z0,tcp\WObj:=Plywood;
    MoveL Offs(pOrigin,116.29,-159.81,-0.00),v40,z0,tcp\WObj:=Plywood;
    MoveL Offs(pOrigin,116.46,-158.64,-0.00),v40,z0,tcp\WObj:=Plywood;
    MoveL Offs(pOrigin,117.00,-157.75,-0.00),v40,z0,tcp\WObj:=Plywood;
    MoveL Offs(pOrigin,116.71,-158.53,-0.00),v40,z0,tcp\WObj:=Plywood;
    MoveL Offs(pOrigin,116.89,-160.55,-0.00),v40,z0,tcp\WObj:=Plywood;
    MoveL Offs(pOrigin,118.13,-162.78,-0.00),v40,z0,tcp\WObj:=Plywood;
    MoveL Offs(pOrigin,119.58,-164.16,-0.00),v40,z0,tcp\WObj:=Plywood;
    MoveL Offs(pOrigin,120.54,-165.97,-0.00),v40,z0,tcp\WObj:=Plywood;
    MoveL Offs(pOrigin,120.64,-167.46,-0.00),v40,z0,tcp\WObj:=Plywood;
    MoveL Offs(pOrigin,120.04,-169.05,-0.00),v40,z0,tcp\WObj:=Plywood;
    MoveL Offs(pOrigin,118.41,-170.15,-0.00),v40,z0,tcp\WObj:=Plywood;
    MoveL Offs(pOrigin,115.12,-170.86,-0.00),v40,z0,tcp\WObj:=Plywood;
    MoveL Offs(pOrigin,109.81,-170.01,-0.00),v40,z0,tcp\WObj:=Plywood;
    MoveL Offs(pOrigin,109.17,-170.22,-0.00),v40,z0,tcp\WObj:=Plywood;
    MoveL Offs(pOrigin,111.61,-170.96,-0.00),v40,z0,tcp\WObj:=Plywood;
    MoveL Offs(pOrigin,113.84,-171.07,-0.00),v40,z0,tcp\WObj:=Plywood;
    MoveL Offs(pOrigin,112.82,-171.28,-0.00),v40,z0,tcp\WObj:=Plywood;
    MoveL Offs(pOrigin,113.63,-171.71,-0.00),v40,z0,tcp\WObj:=Plywood;
    MoveL Offs(pOrigin,117.24,-171.71,-0.00),v40,z0,tcp\WObj:=Plywood;
    MoveL Offs(pOrigin,120.64,-170.47,-0.00),v40,z0,tcp\WObj:=Plywood;
    MoveL Offs(pOrigin,121.71,-169.16,-0.00),v40,z0,tcp\WObj:=Plywood;
    MoveL Offs(pOrigin,122.34,-167.56,-0.00),v40,z0,tcp\WObj:=Plywood;
    MoveL Offs(pOrigin,122.20,-166.61,-0.00),v40,z0,tcp\WObj:=Plywood;
    MoveL Offs(pOrigin,121.07,-164.80,-0.00),v40,z0,tcp\WObj:=Plywood;
    MoveL Offs(pOrigin,118.62,-162.68,-0.00),v40,z0,tcp\WObj:=Plywood;
    MoveL Offs(pOrigin,117.46,-160.34,-0.00),v40,z0,tcp\WObj:=Plywood;
    MoveL Offs(pOrigin,117.46,-158.64,-0.00),v40,z0,tcp\WObj:=Plywood;
    MoveL Offs(pOrigin,118.31,-157.43,-0.00),v40,z0,tcp\WObj:=Plywood;
    MoveL Offs(pOrigin,117.78,-158.64,-0.00),v40,z0,tcp\WObj:=Plywood;
    MoveL Offs(pOrigin,118.16,-160.87,-0.00),v40,z0,tcp\WObj:=Plywood;
    MoveL Offs(pOrigin,118.59,-161.19,-0.00),v40,z0,tcp\WObj:=Plywood;
    MoveL Offs(pOrigin,118.31,-159.06,-0.00),v40,z0,tcp\WObj:=Plywood;
    MoveL Offs(pOrigin,119.12,-157.65,-0.00),v40,z0,tcp\WObj:=Plywood;
    MoveL Offs(pOrigin,118.62,-158.96,-0.00),v40,z0,tcp\WObj:=Plywood;
    MoveL Offs(pOrigin,118.91,-161.08,-0.00),v40,z0,tcp\WObj:=Plywood;
    MoveL Offs(pOrigin,119.58,-162.14,-0.00),v40,z0,tcp\WObj:=Plywood;
    MoveL Offs(pOrigin,121.81,-164.23,-0.00),v40,z0,tcp\WObj:=Plywood;
    MoveL Offs(pOrigin,121.81,-163.84,-0.00),v40,z0,tcp\WObj:=Plywood;
    MoveL Offs(pOrigin,119.65,-161.40,-0.00),v40,z0,tcp\WObj:=Plywood;
    MoveL Offs(pOrigin,119.26,-160.34,-0.00),v40,z0,tcp\WObj:=Plywood;
    MoveL Offs(pOrigin,119.37,-158.64,-0.00),v40,z0,tcp\WObj:=Plywood;
    MoveL Offs(pOrigin,120.11,-157.50,-0.00),v40,z0,tcp\WObj:=Plywood;
    MoveL Offs(pOrigin,119.69,-159.81,-0.00),v40,z0,tcp\WObj:=Plywood;
    MoveL Offs(pOrigin,120.75,-161.72,-0.00),v40,z0,tcp\WObj:=Plywood;
    MoveL Offs(pOrigin,121.21,-161.82,-0.00),v40,z0,tcp\WObj:=Plywood;
    MoveL Offs(pOrigin,120.54,-160.02,-0.00),v40,z0,tcp\WObj:=Plywood;
    MoveL Offs(pOrigin,120.75,-158.39,-0.00),v40,z0,tcp\WObj:=Plywood;
    MoveL Offs(pOrigin,120.96,-158.74,-0.00),v40,z0,tcp\WObj:=Plywood;
    MoveL Offs(pOrigin,121.35,-158.18,-0.00),v40,z0,tcp\WObj:=Plywood;
    MoveL Offs(pOrigin,121.25,-160.23,-0.00),v40,z0,tcp\WObj:=Plywood;
    MoveL Offs(pOrigin,121.92,-161.40,-0.00),v40,z0,tcp\WObj:=Plywood;
    MoveL Offs(pOrigin,122.63,-161.82,-0.00),v40,z0,tcp\WObj:=Plywood;
    MoveL Offs(pOrigin,122.03,-160.34,-0.00),v40,z0,tcp\WObj:=Plywood;
    MoveL Offs(pOrigin,122.03,-159.06,-0.00),v40,z0,tcp\WObj:=Plywood;
    MoveL Offs(pOrigin,122.73,-157.96,-0.00),v40,z0,tcp\WObj:=Plywood;
    MoveL Offs(pOrigin,122.45,-159.38,-0.00),v40,z0,tcp\WObj:=Plywood;
    MoveL Offs(pOrigin,123.19,-161.19,-0.00),v40,z0,tcp\WObj:=Plywood;
    MoveL Offs(pOrigin,124.57,-162.00,-0.00),v40,z0,tcp\WObj:=Plywood;
    MoveL Offs(pOrigin,123.41,-160.23,-0.00),v40,z0,tcp\WObj:=Plywood;
    MoveL Offs(pOrigin,123.30,-158.96,-0.00),v40,z0,tcp\WObj:=Plywood;
    MoveL Offs(pOrigin,123.58,-158.35,-0.00),v40,z0,tcp\WObj:=Plywood;
    MoveL Offs(pOrigin,123.80,-160.12,-0.00),v40,z0,tcp\WObj:=Plywood;
    MoveL Offs(pOrigin,124.68,-161.40,-0.00),v40,z0,tcp\WObj:=Plywood;
    MoveL Offs(pOrigin,127.97,-163.81,-0.00),v40,z0,tcp\WObj:=Plywood;
    MoveL Offs(pOrigin,128.15,-163.63,-0.00),v40,z0,tcp\WObj:=Plywood;
    MoveL Offs(pOrigin,125.74,-161.93,-0.00),v40,z0,tcp\WObj:=Plywood;
    MoveL Offs(pOrigin,124.82,-160.76,-0.00),v40,z0,tcp\WObj:=Plywood;
    MoveL Offs(pOrigin,124.47,-159.70,-0.00),v40,z0,tcp\WObj:=Plywood;
    MoveL Offs(pOrigin,124.75,-158.50,-0.00),v40,z0,tcp\WObj:=Plywood;
    MoveL Offs(pOrigin,125.07,-160.12,-0.00),v40,z0,tcp\WObj:=Plywood;
    MoveL Offs(pOrigin,126.06,-161.36,-0.00),v40,z0,tcp\WObj:=Plywood;
    MoveL Offs(pOrigin,126.24,-161.19,-0.00),v40,z0,tcp\WObj:=Plywood;
    MoveL Offs(pOrigin,125.43,-159.27,-0.00),v40,z0,tcp\WObj:=Plywood;
    MoveL Offs(pOrigin,125.57,-158.35,-0.00),v40,z0,tcp\WObj:=Plywood;
    MoveL Offs(pOrigin,125.96,-159.59,-0.00),v40,z0,tcp\WObj:=Plywood;
  ENDPROC

  PROC DrawPart17()
    MoveL Offs(pOrigin,126.10,-158.71,-0.00),v40,z0,tcp\WObj:=Plywood;
    MoveL Offs(pOrigin,127.23,-160.51,-0.00),v40,z0,tcp\WObj:=Plywood;
    MoveL Offs(pOrigin,128.93,-161.75,-0.00),v40,z0,tcp\WObj:=Plywood;
    MoveL Offs(pOrigin,132.33,-163.45,-0.00),v40,z0,tcp\WObj:=Plywood;
    MoveL Offs(pOrigin,132.23,-162.99,-0.00),v40,z0,tcp\WObj:=Plywood;
    MoveL Offs(pOrigin,130.95,-162.11,-0.00),v40,z0,tcp\WObj:=Plywood;
    MoveL Offs(pOrigin,128.08,-160.76,-0.00),v40,z0,tcp\WObj:=Plywood;
    MoveL Offs(pOrigin,126.31,-158.25,-0.00),v40,z0,tcp\WObj:=Plywood;
    MoveL Offs(pOrigin,126.91,-158.99,-0.00),v40,z0,tcp\WObj:=Plywood;
    MoveL Offs(pOrigin,126.91,-158.18,-0.00),v40,z0,tcp\WObj:=Plywood;
    MoveL Offs(pOrigin,128.51,-159.95,-0.00),v40,z0,tcp\WObj:=Plywood;
    MoveL Offs(pOrigin,131.27,-160.76,-0.00),v40,z0,tcp\WObj:=Plywood;
    MoveL Offs(pOrigin,131.27,-160.51,-0.00),v40,z0,tcp\WObj:=Plywood;
    MoveL Offs(pOrigin,128.61,-159.27,-0.00),v40,z0,tcp\WObj:=Plywood;
    MoveL Offs(pOrigin,128.01,-158.04,-0.00),v40,z0,tcp\WObj:=Plywood;
    MoveL Offs(pOrigin,131.06,-159.70,-0.00),v40,z0,tcp\WObj:=Plywood;
    MoveL Offs(pOrigin,134.14,-160.02,-0.00),v40,z0,tcp\WObj:=Plywood;
    MoveL Offs(pOrigin,134.03,-159.70,-0.00),v40,z0,tcp\WObj:=Plywood;
    MoveL Offs(pOrigin,130.52,-159.03,-0.00),v40,z0,tcp\WObj:=Plywood;
    MoveL Offs(pOrigin,128.97,-157.61,-0.00),v40,z0,tcp\WObj:=Plywood;
    MoveL Offs(pOrigin,131.16,-158.64,-0.00),v40,z0,tcp\WObj:=Plywood;
    MoveL Offs(pOrigin,133.39,-158.74,-0.00),v40,z0,tcp\WObj:=Plywood;
    MoveL Offs(pOrigin,133.29,-158.46,-0.00),v40,z0,tcp\WObj:=Plywood;
    MoveL Offs(pOrigin,131.59,-158.14,-0.00),v40,z0,tcp\WObj:=Plywood;
    MoveL Offs(pOrigin,130.45,-157.33,-0.00),v40,z0,tcp\WObj:=Plywood;
    MoveL Offs(pOrigin,130.84,-157.19,-0.00),v40,z0,tcp\WObj:=Plywood;
    MoveL Offs(pOrigin,133.07,-157.89,-0.00),v40,z0,tcp\WObj:=Plywood;
    MoveL Offs(pOrigin,138.39,-157.57,-0.00),v40,z0,tcp\WObj:=Plywood;
    MoveL Offs(pOrigin,141.47,-158.53,-0.00),v40,z0,tcp\WObj:=Plywood;
    MoveL Offs(pOrigin,142.74,-158.35,-0.00),v40,z0,tcp\WObj:=Plywood;
    MoveL Offs(pOrigin,143.91,-157.57,-0.00),v40,z0,tcp\WObj:=Plywood;
    MoveL Offs(pOrigin,145.40,-154.71,-0.00),v40,z0,tcp\WObj:=Plywood;
    MoveL Offs(pOrigin,146.60,-153.75,-0.00),v40,z0,tcp\WObj:=Plywood;
    MoveL Offs(pOrigin,145.93,-153.64,-0.00),v40,z0,tcp\WObj:=Plywood;
    MoveL Offs(pOrigin,145.19,-154.07,-0.00),v40,z0,tcp\WObj:=Plywood;
    MoveL Offs(pOrigin,144.41,-155.13,-0.00),v40,z0,tcp\WObj:=Plywood;
    MoveL Offs(pOrigin,143.63,-157.15,-0.00),v40,z0,tcp\WObj:=Plywood;
    MoveL Offs(pOrigin,142.92,-157.40,-0.00),v40,z0,tcp\WObj:=Plywood;
    MoveL Offs(pOrigin,143.77,-155.45,-0.00),v40,z0,tcp\WObj:=Plywood;
    MoveL Offs(pOrigin,143.13,-155.95,-0.00),v40,z0,tcp\WObj:=Plywood;
    MoveL Offs(pOrigin,144.12,-154.07,-0.00),v40,z0,tcp\WObj:=Plywood;
    MoveL Offs(pOrigin,143.91,-153.89,-0.00),v40,z0,tcp\WObj:=Plywood;
    MoveL Offs(pOrigin,143.56,-154.18,-0.00),v40,z0,tcp\WObj:=Plywood;
    MoveL Offs(pOrigin,144.55,-152.90,-0.00),v40,z0,tcp\WObj:=Plywood;
    MoveL Offs(pOrigin,145.40,-152.37,-0.00),v40,z0,tcp\WObj:=Plywood;
    MoveL Offs(pOrigin,145.29,-152.05,-0.00),v40,z0,tcp\WObj:=Plywood;
    MoveL Offs(pOrigin,144.34,-152.26,-0.00),v40,z0,tcp\WObj:=Plywood;
    MoveL Offs(pOrigin,141.26,-154.85,-0.00),v40,z0,tcp\WObj:=Plywood;
    MoveL Offs(pOrigin,137.54,-155.88,-0.00),v40,z0,tcp\WObj:=Plywood;
    MoveL Offs(pOrigin,138.60,-156.09,-0.00),v40,z0,tcp\WObj:=Plywood;
    MoveL Offs(pOrigin,142.04,-155.20,-0.00),v40,z0,tcp\WObj:=Plywood;
    MoveL Offs(pOrigin,139.52,-156.30,-0.00),v40,z0,tcp\WObj:=Plywood;
    MoveL Offs(pOrigin,141.61,-156.62,-0.00),v40,z0,tcp\WObj:=Plywood;
    MoveL Offs(pOrigin,138.99,-156.83,-0.00),v40,z0,tcp\WObj:=Plywood;
    MoveL Offs(pOrigin,140.87,-157.47,-0.00),v40,z0,tcp\WObj:=Plywood;
    MoveL Offs(pOrigin,138.28,-157.04,-0.00),v40,z0,tcp\WObj:=Plywood;
    MoveL Offs(pOrigin,133.39,-157.36,-0.00),v40,z0,tcp\WObj:=Plywood;
    MoveL Offs(pOrigin,132.40,-156.87,-0.00),v40,z0,tcp\WObj:=Plywood;
    MoveL Offs(pOrigin,133.71,-156.94,-0.00),v40,z0,tcp\WObj:=Plywood;
    MoveL Offs(pOrigin,136.26,-156.44,-0.00),v40,z0,tcp\WObj:=Plywood;
    MoveL Offs(pOrigin,136.26,-156.19,-0.00),v40,z0,tcp\WObj:=Plywood;
    MoveL Offs(pOrigin,133.78,-156.30,-0.00),v40,z0,tcp\WObj:=Plywood;
    MoveL Offs(pOrigin,136.79,-155.49,-0.00),v40,z0,tcp\WObj:=Plywood;
    MoveL Offs(pOrigin,137.96,-154.81,-0.00),v40,z0,tcp\WObj:=Plywood;
    MoveL Offs(pOrigin,137.86,-154.60,-0.00),v40,z0,tcp\WObj:=Plywood;
    MoveL Offs(pOrigin,135.48,-155.10,-0.00),v40,z0,tcp\WObj:=Plywood;
    MoveL Offs(pOrigin,137.54,-154.18,-0.00),v40,z0,tcp\WObj:=Plywood;
    MoveL Offs(pOrigin,137.75,-153.79,-0.00),v40,z0,tcp\WObj:=Plywood;
    MoveL Offs(pOrigin,136.44,-154.28,-0.00),v40,z0,tcp\WObj:=Plywood;
    MoveL Offs(pOrigin,138.60,-152.79,-0.00),v40,z0,tcp\WObj:=Plywood;
    MoveL Offs(pOrigin,138.71,-152.30,-0.00),v40,z0,tcp\WObj:=Plywood;
    MoveL Offs(pOrigin,137.82,-152.97,-0.00),v40,z0,tcp\WObj:=Plywood;
    MoveL Offs(pOrigin,140.55,-150.14,-0.00),v40,z0,tcp\WObj:=Plywood;
    MoveL Offs(pOrigin,140.30,-150.03,-0.00),v40,z0,tcp\WObj:=Plywood;
    MoveL Offs(pOrigin,138.25,-151.70,-0.00),v40,z0,tcp\WObj:=Plywood;
    MoveL Offs(pOrigin,139.45,-150.35,-0.00),v40,z0,tcp\WObj:=Plywood;
    MoveL Offs(pOrigin,139.10,-150.31,-0.00),v40,z0,tcp\WObj:=Plywood;
    MoveL Offs(pOrigin,140.69,-148.01,-0.00),v40,z0,tcp\WObj:=Plywood;
    MoveL Offs(pOrigin,139.27,-149.22,-0.00),v40,z0,tcp\WObj:=Plywood;
    MoveL Offs(pOrigin,140.90,-146.95,-0.00),v40,z0,tcp\WObj:=Plywood;
    MoveL Offs(pOrigin,139.49,-148.05,-0.00),v40,z0,tcp\WObj:=Plywood;
    MoveL Offs(pOrigin,141.01,-145.36,-0.00),v40,z0,tcp\WObj:=Plywood;
    MoveL Offs(pOrigin,139.31,-146.95,-0.00),v40,z0,tcp\WObj:=Plywood;
    MoveL Offs(pOrigin,143.38,-141.53,-0.00),v40,z0,tcp\WObj:=Plywood;
    MoveL Offs(pOrigin,144.98,-140.61,-0.00),v40,z0,tcp\WObj:=Plywood;
    MoveL Offs(pOrigin,144.80,-141.11,-0.00),v40,z0,tcp\WObj:=Plywood;
    MoveL Offs(pOrigin,146.82,-141.43,-0.00),v40,z0,tcp\WObj:=Plywood;
    MoveL Offs(pOrigin,145.72,-140.89,-0.00),v40,z0,tcp\WObj:=Plywood;
    MoveL Offs(pOrigin,144.80,-141.11,-0.00),v40,z0,tcp\WObj:=Plywood;
    MoveL Offs(pOrigin,144.34,-141.35,-0.00),v40,z0,tcp\WObj:=Plywood;
    MoveL Offs(pOrigin,143.27,-142.06,-0.00),v40,z0,tcp\WObj:=Plywood;
    MoveL Offs(pOrigin,145.61,-141.96,-0.00),v40,z0,tcp\WObj:=Plywood;
    MoveL Offs(pOrigin,148.13,-143.23,-0.00),v40,z0,tcp\WObj:=Plywood;
    MoveL Offs(pOrigin,147.31,-142.17,-0.00),v40,z0,tcp\WObj:=Plywood;
    MoveL Offs(pOrigin,145.82,-141.53,-0.00),v40,z0,tcp\WObj:=Plywood;
    MoveL Offs(pOrigin,144.34,-141.35,-0.00),v40,fine,tcp\WObj:=Plywood;
    MoveL Offs(pOrigin,144.34,-141.35,-6.00),v60,z5,tcp\WObj:=Plywood;
    MoveL Offs(pOrigin,145.08,-142.38,-6.00),vTravel,z5,tcp\WObj:=Plywood;
    MoveL Offs(pOrigin,145.08,-142.38,-0.00),v60,z0,tcp\WObj:=Plywood;
    MoveL Offs(pOrigin,143.98,-142.81,-0.00),v40,z0,tcp\WObj:=Plywood;
    MoveL Offs(pOrigin,145.82,-142.91,-0.00),v40,z0,tcp\WObj:=Plywood;
    MoveL Offs(pOrigin,148.02,-143.98,-0.00),v40,z0,tcp\WObj:=Plywood;
    MoveL Offs(pOrigin,147.42,-143.23,-0.00),v40,z0,tcp\WObj:=Plywood;
    MoveL Offs(pOrigin,145.93,-142.49,-0.00),v40,z0,tcp\WObj:=Plywood;
    MoveL Offs(pOrigin,145.08,-142.38,-0.00),v40,z0,tcp\WObj:=Plywood;
    MoveL Offs(pOrigin,144.90,-143.23,-0.00),v40,z0,tcp\WObj:=Plywood;
    MoveL Offs(pOrigin,143.17,-143.41,-0.00),v40,z0,tcp\WObj:=Plywood;
    MoveL Offs(pOrigin,141.82,-144.72,-0.00),v40,z0,tcp\WObj:=Plywood;
    MoveL Offs(pOrigin,144.90,-143.23,-0.00),v40,z0,tcp\WObj:=Plywood;
    MoveL Offs(pOrigin,145.29,-143.66,-0.00),v40,z0,tcp\WObj:=Plywood;
    MoveL Offs(pOrigin,143.81,-144.05,-0.00),v40,z0,tcp\WObj:=Plywood;
    MoveL Offs(pOrigin,142.32,-144.93,-0.00),v40,z0,tcp\WObj:=Plywood;
    MoveL Offs(pOrigin,140.87,-146.74,-0.00),v40,z0,tcp\WObj:=Plywood;
    MoveL Offs(pOrigin,142.85,-145.11,-0.00),v40,z0,tcp\WObj:=Plywood;
    MoveL Offs(pOrigin,145.08,-144.40,-0.00),v40,z0,tcp\WObj:=Plywood;
    MoveL Offs(pOrigin,146.57,-144.68,-0.00),v40,z0,tcp\WObj:=Plywood;
    MoveL Offs(pOrigin,147.63,-145.46,-0.00),v40,z0,tcp\WObj:=Plywood;
    MoveL Offs(pOrigin,148.16,-146.31,-0.00),v40,z0,tcp\WObj:=Plywood;
    MoveL Offs(pOrigin,148.38,-146.21,-0.00),v40,z0,tcp\WObj:=Plywood;
    MoveL Offs(pOrigin,147.52,-144.72,-0.00),v40,z0,tcp\WObj:=Plywood;
  ENDPROC

  PROC DrawPart18()
    MoveL Offs(pOrigin,146.57,-144.01,-0.00),v40,z0,tcp\WObj:=Plywood;
    MoveL Offs(pOrigin,145.29,-143.66,-0.00),v40,fine,tcp\WObj:=Plywood;
    MoveL Offs(pOrigin,145.29,-143.66,-6.00),v60,z5,tcp\WObj:=Plywood;
    MoveL Offs(pOrigin,144.98,-144.93,-6.00),vTravel,z5,tcp\WObj:=Plywood;
    MoveL Offs(pOrigin,144.98,-144.93,-0.00),v60,z0,tcp\WObj:=Plywood;
    MoveL Offs(pOrigin,143.88,-145.46,-0.00),v40,z0,tcp\WObj:=Plywood;
    MoveL Offs(pOrigin,145.72,-145.46,-0.00),v40,z0,tcp\WObj:=Plywood;
    MoveL Offs(pOrigin,147.84,-146.31,-0.00),v40,z0,tcp\WObj:=Plywood;
    MoveL Offs(pOrigin,147.10,-145.46,-0.00),v40,z0,tcp\WObj:=Plywood;
    MoveL Offs(pOrigin,145.93,-144.93,-0.00),v40,z0,tcp\WObj:=Plywood;
    MoveL Offs(pOrigin,144.98,-144.93,-0.00),v40,z0,tcp\WObj:=Plywood;
    MoveL Offs(pOrigin,144.66,-145.68,-0.00),v40,z0,tcp\WObj:=Plywood;
    MoveL Offs(pOrigin,142.96,-146.28,-0.00),v40,z0,tcp\WObj:=Plywood;
    MoveL Offs(pOrigin,141.36,-147.91,-0.00),v40,z0,tcp\WObj:=Plywood;
    MoveL Offs(pOrigin,140.76,-149.18,-0.00),v40,z0,tcp\WObj:=Plywood;
    MoveL Offs(pOrigin,143.59,-146.70,-0.00),v40,z0,tcp\WObj:=Plywood;
    MoveL Offs(pOrigin,145.93,-145.89,-0.00),v40,z0,tcp\WObj:=Plywood;
    MoveL Offs(pOrigin,144.66,-145.68,-0.00),v40,z0,tcp\WObj:=Plywood;
    MoveL Offs(pOrigin,144.98,-146.74,-0.00),v40,z0,tcp\WObj:=Plywood;
    MoveL Offs(pOrigin,143.56,-147.48,-0.00),v40,z0,tcp\WObj:=Plywood;
    MoveL Offs(pOrigin,145.82,-147.27,-0.00),v40,z0,tcp\WObj:=Plywood;
    MoveL Offs(pOrigin,147.88,-148.12,-0.00),v40,z0,tcp\WObj:=Plywood;
    MoveL Offs(pOrigin,147.21,-147.27,-0.00),v40,z0,tcp\WObj:=Plywood;
    MoveL Offs(pOrigin,146.04,-146.74,-0.00),v40,z0,tcp\WObj:=Plywood;
    MoveL Offs(pOrigin,144.98,-146.74,-0.00),v40,z0,tcp\WObj:=Plywood;
    MoveL Offs(pOrigin,144.55,-147.62,-0.00),v40,z0,tcp\WObj:=Plywood;
    MoveL Offs(pOrigin,142.96,-148.05,-0.00),v40,z0,tcp\WObj:=Plywood;
    MoveL Offs(pOrigin,141.79,-148.86,-0.00),v40,z0,tcp\WObj:=Plywood;
    MoveL Offs(pOrigin,140.76,-150.14,-0.00),v40,z0,tcp\WObj:=Plywood;
    MoveL Offs(pOrigin,142.32,-148.83,-0.00),v40,z0,tcp\WObj:=Plywood;
    MoveL Offs(pOrigin,144.55,-147.62,-0.00),v40,fine,tcp\WObj:=Plywood;
    MoveL Offs(pOrigin,144.55,-147.62,-6.00),v60,z5,tcp\WObj:=Plywood;
    MoveL Offs(pOrigin,145.51,-148.54,-6.00),vTravel,z5,tcp\WObj:=Plywood;
    MoveL Offs(pOrigin,145.51,-148.54,-0.00),v60,z0,tcp\WObj:=Plywood;
    MoveL Offs(pOrigin,146.78,-148.76,-0.00),v40,z0,tcp\WObj:=Plywood;
    MoveL Offs(pOrigin,146.89,-148.54,-0.00),v40,z0,tcp\WObj:=Plywood;
    MoveL Offs(pOrigin,145.82,-148.01,-0.00),v40,z0,tcp\WObj:=Plywood;
    MoveL Offs(pOrigin,143.49,-148.51,-0.00),v40,z0,tcp\WObj:=Plywood;
    MoveL Offs(pOrigin,142.21,-149.39,-0.00),v40,z0,tcp\WObj:=Plywood;
    MoveL Offs(pOrigin,139.80,-152.16,-0.00),v40,z0,tcp\WObj:=Plywood;
    MoveL Offs(pOrigin,143.17,-149.46,-0.00),v40,z0,tcp\WObj:=Plywood;
    MoveL Offs(pOrigin,145.51,-148.54,-0.00),v40,z0,tcp\WObj:=Plywood;
    MoveL Offs(pOrigin,145.19,-149.39,-0.00),v40,z0,tcp\WObj:=Plywood;
    MoveL Offs(pOrigin,143.98,-150.03,-0.00),v40,z0,tcp\WObj:=Plywood;
    MoveL Offs(pOrigin,145.93,-149.93,-0.00),v40,z0,tcp\WObj:=Plywood;
    MoveL Offs(pOrigin,147.91,-150.67,-0.00),v40,z0,tcp\WObj:=Plywood;
    MoveL Offs(pOrigin,147.42,-149.93,-0.00),v40,z0,tcp\WObj:=Plywood;
    MoveL Offs(pOrigin,146.36,-149.39,-0.00),v40,z0,tcp\WObj:=Plywood;
    MoveL Offs(pOrigin,145.19,-149.39,-0.00),v40,z0,tcp\WObj:=Plywood;
    MoveL Offs(pOrigin,144.87,-150.14,-0.00),v40,z0,tcp\WObj:=Plywood;
    MoveL Offs(pOrigin,143.38,-150.74,-0.00),v40,z0,tcp\WObj:=Plywood;
    MoveL Offs(pOrigin,138.81,-154.88,-0.00),v40,z0,tcp\WObj:=Plywood;
    MoveL Offs(pOrigin,139.77,-154.53,-0.00),v40,z0,tcp\WObj:=Plywood;
    MoveL Offs(pOrigin,142.96,-152.37,-0.00),v40,z0,tcp\WObj:=Plywood;
    MoveL Offs(pOrigin,144.23,-151.09,-0.00),v40,z0,tcp\WObj:=Plywood;
    MoveL Offs(pOrigin,145.82,-150.28,-0.00),v40,z0,tcp\WObj:=Plywood;
    MoveL Offs(pOrigin,144.87,-150.14,-0.00),v40,z0,tcp\WObj:=Plywood;
    MoveL Offs(pOrigin,145.72,-150.95,-0.00),v40,z0,tcp\WObj:=Plywood;
    MoveL Offs(pOrigin,139.41,-154.92,-0.00),v40,z0,tcp\WObj:=Plywood;
    MoveL Offs(pOrigin,141.47,-154.42,-0.00),v40,z0,tcp\WObj:=Plywood;
    MoveL Offs(pOrigin,143.91,-152.30,-0.00),v40,z0,tcp\WObj:=Plywood;
    MoveL Offs(pOrigin,146.46,-151.80,-0.00),v40,z0,tcp\WObj:=Plywood;
    MoveL Offs(pOrigin,146.14,-151.34,-0.00),v40,z0,tcp\WObj:=Plywood;
    MoveL Offs(pOrigin,147.84,-151.98,-0.00),v40,z0,tcp\WObj:=Plywood;
    MoveL Offs(pOrigin,147.91,-151.73,-0.00),v40,z0,tcp\WObj:=Plywood;
    MoveL Offs(pOrigin,147.10,-150.95,-0.00),v40,z0,tcp\WObj:=Plywood;
    MoveL Offs(pOrigin,145.72,-150.95,-0.00),v40,fine,tcp\WObj:=Plywood;
    MoveL Offs(pOrigin,145.72,-150.95,-6.00),v60,z5,tcp\WObj:=Plywood;
    MoveL Offs(pOrigin,146.04,-152.79,-6.00),vTravel,z5,tcp\WObj:=Plywood;
    MoveL Offs(pOrigin,146.04,-152.79,-0.00),v60,z0,tcp\WObj:=Plywood;
    MoveL Offs(pOrigin,144.80,-153.75,-0.00),v40,z0,tcp\WObj:=Plywood;
    MoveL Offs(pOrigin,146.14,-153.22,-0.00),v40,z0,tcp\WObj:=Plywood;
    MoveL Offs(pOrigin,147.70,-153.32,-0.00),v40,z0,tcp\WObj:=Plywood;
    MoveL Offs(pOrigin,146.99,-152.79,-0.00),v40,z0,tcp\WObj:=Plywood;
    MoveL Offs(pOrigin,146.04,-152.79,-0.00),v40,z0,tcp\WObj:=Plywood;
    MoveL Offs(pOrigin,147.10,-152.40,-0.00),v40,z0,tcp\WObj:=Plywood;
    MoveL Offs(pOrigin,147.52,-152.76,-0.00),v40,z0,tcp\WObj:=Plywood;
    MoveL Offs(pOrigin,147.10,-152.40,-0.00),v40,fine,tcp\WObj:=Plywood;
    MoveL Offs(pOrigin,147.10,-152.40,-6.00),v60,z5,tcp\WObj:=Plywood;
    MoveL Offs(pOrigin,147.42,-154.56,-6.00),vTravel,z5,tcp\WObj:=Plywood;
    MoveL Offs(pOrigin,147.42,-154.56,-0.00),v60,z0,tcp\WObj:=Plywood;
    MoveL Offs(pOrigin,147.21,-155.49,-0.00),v40,z0,tcp\WObj:=Plywood;
    MoveL Offs(pOrigin,147.60,-154.81,-0.00),v40,z0,tcp\WObj:=Plywood;
    MoveL Offs(pOrigin,147.42,-154.56,-0.00),v40,fine,tcp\WObj:=Plywood;
    MoveL Offs(pOrigin,147.42,-154.56,-6.00),v60,z5,tcp\WObj:=Plywood;
    MoveL Offs(pOrigin,146.14,-155.52,-6.00),vTravel,z5,tcp\WObj:=Plywood;
    MoveL Offs(pOrigin,146.14,-155.52,-0.00),v60,z0,tcp\WObj:=Plywood;
    MoveL Offs(pOrigin,146.04,-156.44,-0.00),v40,z0,tcp\WObj:=Plywood;
    MoveL Offs(pOrigin,146.43,-155.88,-0.00),v40,z0,tcp\WObj:=Plywood;
    MoveL Offs(pOrigin,146.14,-155.52,-0.00),v40,z0,tcp\WObj:=Plywood;
    MoveL Offs(pOrigin,145.51,-156.41,-0.00),v40,z0,tcp\WObj:=Plywood;
    MoveL Offs(pOrigin,143.59,-158.96,-0.00),v40,z0,tcp\WObj:=Plywood;
    MoveL Offs(pOrigin,142.00,-159.70,-0.00),v40,z0,tcp\WObj:=Plywood;
    MoveL Offs(pOrigin,140.62,-159.59,-0.00),v40,z0,tcp\WObj:=Plywood;
    MoveL Offs(pOrigin,137.96,-158.43,-0.00),v40,z0,tcp\WObj:=Plywood;
    MoveL Offs(pOrigin,135.80,-158.53,-0.00),v40,z0,tcp\WObj:=Plywood;
    MoveL Offs(pOrigin,139.38,-159.70,-0.00),v40,z0,tcp\WObj:=Plywood;
    MoveL Offs(pOrigin,138.71,-159.81,-0.00),v40,z0,tcp\WObj:=Plywood;
    MoveL Offs(pOrigin,139.88,-160.48,-0.00),v40,z0,tcp\WObj:=Plywood;
    MoveL Offs(pOrigin,142.21,-160.87,-0.00),v40,z0,tcp\WObj:=Plywood;
    MoveL Offs(pOrigin,143.27,-160.44,-0.00),v40,z0,tcp\WObj:=Plywood;
    MoveL Offs(pOrigin,144.34,-159.38,-0.00),v40,z0,tcp\WObj:=Plywood;
    MoveL Offs(pOrigin,145.12,-158.00,-0.00),v40,z0,tcp\WObj:=Plywood;
    MoveL Offs(pOrigin,145.51,-156.41,-0.00),v40,fine,tcp\WObj:=Plywood;
    MoveL Offs(pOrigin,145.51,-156.41,-6.00),v60,z5,tcp\WObj:=Plywood;
    MoveL Offs(pOrigin,143.84,-158.00,-6.00),vTravel,z5,tcp\WObj:=Plywood;
    MoveL Offs(pOrigin,143.84,-158.00,-0.00),v60,z0,tcp\WObj:=Plywood;
    MoveL Offs(pOrigin,141.68,-158.74,-0.00),v40,z0,tcp\WObj:=Plywood;
    MoveL Offs(pOrigin,138.60,-158.11,-0.00),v40,z0,tcp\WObj:=Plywood;
    MoveL Offs(pOrigin,138.42,-158.32,-0.00),v40,z0,tcp\WObj:=Plywood;
    MoveL Offs(pOrigin,140.09,-159.20,-0.00),v40,z0,tcp\WObj:=Plywood;
    MoveL Offs(pOrigin,141.79,-159.49,-0.00),v40,z0,tcp\WObj:=Plywood;
    MoveL Offs(pOrigin,143.38,-158.64,-0.00),v40,z0,tcp\WObj:=Plywood;
    MoveL Offs(pOrigin,143.84,-158.00,-0.00),v40,fine,tcp\WObj:=Plywood;
    MoveL Offs(pOrigin,143.84,-158.00,-6.00),v60,z5,tcp\WObj:=Plywood;
    MoveL Offs(pOrigin,144.76,-159.52,-6.00),vTravel,z5,tcp\WObj:=Plywood;
    MoveL Offs(pOrigin,144.76,-159.52,-0.00),v60,z0,tcp\WObj:=Plywood;
    MoveL Offs(pOrigin,142.85,-160.90,-0.00),v40,z0,tcp\WObj:=Plywood;
    MoveL Offs(pOrigin,141.15,-161.08,-0.00),v40,z0,tcp\WObj:=Plywood;
    MoveL Offs(pOrigin,136.79,-159.49,-0.00),v40,z0,tcp\WObj:=Plywood;
  ENDPROC

  PROC DrawPart19()
    MoveL Offs(pOrigin,134.21,-159.38,-0.00),v40,z0,tcp\WObj:=Plywood;
    MoveL Offs(pOrigin,136.90,-160.20,-0.00),v40,z0,tcp\WObj:=Plywood;
    MoveL Offs(pOrigin,139.66,-161.97,-0.00),v40,z0,tcp\WObj:=Plywood;
    MoveL Offs(pOrigin,140.83,-162.36,-0.00),v40,z0,tcp\WObj:=Plywood;
    MoveL Offs(pOrigin,142.96,-161.86,-0.00),v40,z0,tcp\WObj:=Plywood;
    MoveL Offs(pOrigin,144.23,-160.76,-0.00),v40,z0,tcp\WObj:=Plywood;
    MoveL Offs(pOrigin,144.90,-159.70,-0.00),v40,z0,tcp\WObj:=Plywood;
    MoveL Offs(pOrigin,144.76,-159.52,-0.00),v40,z0,tcp\WObj:=Plywood;
    MoveL Offs(pOrigin,145.72,-158.89,-0.00),v40,z0,tcp\WObj:=Plywood;
    MoveL Offs(pOrigin,145.82,-158.39,-0.00),v40,z0,tcp\WObj:=Plywood;
    MoveL Offs(pOrigin,145.72,-158.89,-0.00),v40,fine,tcp\WObj:=Plywood;
    MoveL Offs(pOrigin,145.72,-158.89,-6.00),v60,z5,tcp\WObj:=Plywood;
    MoveL Offs(pOrigin,144.12,-161.82,-6.00),vTravel,z5,tcp\WObj:=Plywood;
    MoveL Offs(pOrigin,144.12,-161.82,-0.00),v60,z0,tcp\WObj:=Plywood;
    MoveL Offs(pOrigin,141.68,-164.48,-0.00),v40,z0,tcp\WObj:=Plywood;
    MoveL Offs(pOrigin,139.77,-165.23,-0.00),v40,z0,tcp\WObj:=Plywood;
    MoveL Offs(pOrigin,137.22,-164.94,-0.00),v40,z0,tcp\WObj:=Plywood;
    MoveL Offs(pOrigin,134.14,-162.75,-0.00),v40,z0,tcp\WObj:=Plywood;
    MoveL Offs(pOrigin,131.98,-162.25,-0.00),v40,z0,tcp\WObj:=Plywood;
    MoveL Offs(pOrigin,135.09,-165.58,-0.00),v40,z0,tcp\WObj:=Plywood;
    MoveL Offs(pOrigin,135.70,-165.76,-0.00),v40,z0,tcp\WObj:=Plywood;
    MoveL Offs(pOrigin,133.11,-162.71,-0.00),v40,z0,tcp\WObj:=Plywood;
    MoveL Offs(pOrigin,135.84,-165.26,-0.00),v40,z0,tcp\WObj:=Plywood;
    MoveL Offs(pOrigin,137.32,-165.86,-0.00),v40,z0,tcp\WObj:=Plywood;
    MoveL Offs(pOrigin,138.60,-165.97,-0.00),v40,z0,tcp\WObj:=Plywood;
    MoveL Offs(pOrigin,140.19,-165.58,-0.00),v40,z0,tcp\WObj:=Plywood;
    MoveL Offs(pOrigin,142.11,-164.59,-0.00),v40,z0,tcp\WObj:=Plywood;
    MoveL Offs(pOrigin,144.34,-161.93,-0.00),v40,z0,tcp\WObj:=Plywood;
    MoveL Offs(pOrigin,144.12,-161.82,-0.00),v40,fine,tcp\WObj:=Plywood;
    MoveL Offs(pOrigin,144.12,-161.82,-6.00),v60,z5,tcp\WObj:=Plywood;
    MoveL Offs(pOrigin,142.78,-162.46,-6.00),vTravel,z5,tcp\WObj:=Plywood;
    MoveL Offs(pOrigin,142.78,-162.46,-0.00),v60,z0,tcp\WObj:=Plywood;
    MoveL Offs(pOrigin,140.51,-162.46,-0.00),v40,z0,tcp\WObj:=Plywood;
    MoveL Offs(pOrigin,137.54,-160.73,-0.00),v40,z0,tcp\WObj:=Plywood;
    MoveL Offs(pOrigin,135.59,-160.34,-0.00),v40,z0,tcp\WObj:=Plywood;
    MoveL Offs(pOrigin,137.79,-161.54,-0.00),v40,z0,tcp\WObj:=Plywood;
    MoveL Offs(pOrigin,135.73,-161.05,-0.00),v40,z0,tcp\WObj:=Plywood;
    MoveL Offs(pOrigin,139.77,-163.31,-0.00),v40,z0,tcp\WObj:=Plywood;
    MoveL Offs(pOrigin,141.15,-163.31,-0.00),v40,z0,tcp\WObj:=Plywood;
    MoveL Offs(pOrigin,142.78,-162.46,-0.00),v40,fine,tcp\WObj:=Plywood;
    MoveL Offs(pOrigin,142.78,-162.46,-6.00),v60,z5,tcp\WObj:=Plywood;
    MoveL Offs(pOrigin,141.65,-163.74,-6.00),vTravel,z5,tcp\WObj:=Plywood;
    MoveL Offs(pOrigin,141.65,-163.74,-0.00),v60,z0,tcp\WObj:=Plywood;
    MoveL Offs(pOrigin,138.92,-163.35,-0.00),v40,z0,tcp\WObj:=Plywood;
    MoveL Offs(pOrigin,134.99,-161.29,-0.00),v40,z0,tcp\WObj:=Plywood;
    MoveL Offs(pOrigin,134.77,-161.47,-0.00),v40,z0,tcp\WObj:=Plywood;
    MoveL Offs(pOrigin,136.65,-162.82,-0.00),v40,z0,tcp\WObj:=Plywood;
    MoveL Offs(pOrigin,134.14,-161.44,-0.00),v40,z0,tcp\WObj:=Plywood;
    MoveL Offs(pOrigin,133.61,-161.61,-0.00),v40,z0,tcp\WObj:=Plywood;
    MoveL Offs(pOrigin,130.06,-160.98,-0.00),v40,z0,tcp\WObj:=Plywood;
    MoveL Offs(pOrigin,130.74,-161.40,-0.00),v40,z0,tcp\WObj:=Plywood;
    MoveL Offs(pOrigin,133.50,-161.97,-0.00),v40,z0,tcp\WObj:=Plywood;
    MoveL Offs(pOrigin,136.48,-164.20,-0.00),v40,z0,tcp\WObj:=Plywood;
    MoveL Offs(pOrigin,138.07,-164.69,-0.00),v40,z0,tcp\WObj:=Plywood;
    MoveL Offs(pOrigin,139.66,-164.69,-0.00),v40,z0,tcp\WObj:=Plywood;
    MoveL Offs(pOrigin,139.73,-164.38,-0.00),v40,z0,tcp\WObj:=Plywood;
    MoveL Offs(pOrigin,141.65,-163.74,-0.00),v40,fine,tcp\WObj:=Plywood;
    MoveL Offs(pOrigin,141.65,-163.74,-6.00),v60,z5,tcp\WObj:=Plywood;
    MoveL Offs(pOrigin,136.94,-166.39,-6.00),vTravel,z5,tcp\WObj:=Plywood;
    MoveL Offs(pOrigin,136.94,-166.39,-0.00),v60,z0,tcp\WObj:=Plywood;
    MoveL Offs(pOrigin,135.98,-166.07,-0.00),v40,z0,tcp\WObj:=Plywood;
    MoveL Offs(pOrigin,136.37,-166.43,-0.00),v40,z0,tcp\WObj:=Plywood;
    MoveL Offs(pOrigin,136.94,-166.39,-0.00),v40,z0,tcp\WObj:=Plywood;
    MoveL Offs(pOrigin,136.58,-166.82,-0.00),v40,z0,tcp\WObj:=Plywood;
    MoveL Offs(pOrigin,136.09,-166.93,-0.00),v40,z0,tcp\WObj:=Plywood;
    MoveL Offs(pOrigin,134.03,-169.05,-0.00),v40,z0,tcp\WObj:=Plywood;
    MoveL Offs(pOrigin,134.03,-169.44,-0.00),v40,z0,tcp\WObj:=Plywood;
    MoveL Offs(pOrigin,135.94,-168.09,-0.00),v40,z0,tcp\WObj:=Plywood;
    MoveL Offs(pOrigin,136.58,-166.82,-0.00),v40,z0,tcp\WObj:=Plywood;
    MoveL Offs(pOrigin,135.73,-166.93,-0.00),v40,z0,tcp\WObj:=Plywood;
    MoveL Offs(pOrigin,135.70,-166.18,-0.00),v40,z0,tcp\WObj:=Plywood;
    MoveL Offs(pOrigin,135.09,-165.76,-0.00),v40,z0,tcp\WObj:=Plywood;
    MoveL Offs(pOrigin,134.99,-167.81,-0.00),v40,z0,tcp\WObj:=Plywood;
    MoveL Offs(pOrigin,135.73,-166.93,-0.00),v40,fine,tcp\WObj:=Plywood;
    MoveL Offs(pOrigin,135.73,-166.93,-6.00),v60,z5,tcp\WObj:=Plywood;
    MoveL Offs(pOrigin,134.77,-165.97,-6.00),vTravel,z5,tcp\WObj:=Plywood;
    MoveL Offs(pOrigin,134.77,-165.97,-0.00),v60,z0,tcp\WObj:=Plywood;
    MoveL Offs(pOrigin,134.24,-165.37,-0.00),v40,z0,tcp\WObj:=Plywood;
    MoveL Offs(pOrigin,134.46,-167.81,-0.00),v40,z0,tcp\WObj:=Plywood;
    MoveL Offs(pOrigin,134.77,-165.97,-0.00),v40,z0,tcp\WObj:=Plywood;
    MoveL Offs(pOrigin,133.82,-165.83,-0.00),v40,z0,tcp\WObj:=Plywood;
    MoveL Offs(pOrigin,133.50,-164.59,-0.00),v40,z0,tcp\WObj:=Plywood;
    MoveL Offs(pOrigin,132.12,-163.52,-0.00),v40,z0,tcp\WObj:=Plywood;
    MoveL Offs(pOrigin,133.82,-165.83,-0.00),v40,z0,tcp\WObj:=Plywood;
    MoveL Offs(pOrigin,133.18,-166.50,-0.00),v40,z0,tcp\WObj:=Plywood;
    MoveL Offs(pOrigin,132.58,-165.01,-0.00),v40,z0,tcp\WObj:=Plywood;
    MoveL Offs(pOrigin,130.42,-162.96,-0.00),v40,z0,tcp\WObj:=Plywood;
    MoveL Offs(pOrigin,130.24,-163.10,-0.00),v40,z0,tcp\WObj:=Plywood;
    MoveL Offs(pOrigin,131.73,-165.23,-0.00),v40,z0,tcp\WObj:=Plywood;
    MoveL Offs(pOrigin,132.01,-167.35,-0.00),v40,z0,tcp\WObj:=Plywood;
    MoveL Offs(pOrigin,131.52,-168.84,-0.00),v40,z0,tcp\WObj:=Plywood;
    MoveL Offs(pOrigin,129.89,-170.79,-0.00),v40,z0,tcp\WObj:=Plywood;
    MoveL Offs(pOrigin,132.40,-169.05,-0.00),v40,z0,tcp\WObj:=Plywood;
    MoveL Offs(pOrigin,133.18,-167.46,-0.00),v40,z0,tcp\WObj:=Plywood;
    MoveL Offs(pOrigin,133.18,-166.50,-0.00),v40,z0,tcp\WObj:=Plywood;
    MoveL Offs(pOrigin,133.71,-167.31,-0.00),v40,z0,tcp\WObj:=Plywood;
    MoveL Offs(pOrigin,132.97,-169.09,-0.00),v40,z0,tcp\WObj:=Plywood;
    MoveL Offs(pOrigin,133.68,-168.31,-0.00),v40,z0,tcp\WObj:=Plywood;
    MoveL Offs(pOrigin,133.71,-167.31,-0.00),v40,fine,tcp\WObj:=Plywood;
    MoveL Offs(pOrigin,133.71,-167.31,-6.00),v60,z5,tcp\WObj:=Plywood;
    MoveL Offs(pOrigin,131.69,-166.50,-6.00),vTravel,z5,tcp\WObj:=Plywood;
    MoveL Offs(pOrigin,131.69,-166.50,-0.00),v60,z0,tcp\WObj:=Plywood;
    MoveL Offs(pOrigin,130.74,-164.38,-0.00),v40,z0,tcp\WObj:=Plywood;
    MoveL Offs(pOrigin,126.59,-161.05,-0.00),v40,z0,tcp\WObj:=Plywood;
    MoveL Offs(pOrigin,126.81,-161.72,-0.00),v40,z0,tcp\WObj:=Plywood;
    MoveL Offs(pOrigin,129.46,-164.16,-0.00),v40,z0,tcp\WObj:=Plywood;
    MoveL Offs(pOrigin,130.42,-166.71,-0.00),v40,z0,tcp\WObj:=Plywood;
    MoveL Offs(pOrigin,129.82,-169.05,-0.00),v40,z0,tcp\WObj:=Plywood;
    MoveL Offs(pOrigin,127.34,-171.56,-0.00),v40,z0,tcp\WObj:=Plywood;
    MoveL Offs(pOrigin,128.40,-171.21,-0.00),v40,z0,tcp\WObj:=Plywood;
    MoveL Offs(pOrigin,130.63,-169.58,-0.00),v40,z0,tcp\WObj:=Plywood;
    MoveL Offs(pOrigin,131.52,-168.09,-0.00),v40,z0,tcp\WObj:=Plywood;
    MoveL Offs(pOrigin,131.69,-166.50,-0.00),v40,fine,tcp\WObj:=Plywood;
    MoveL Offs(pOrigin,131.69,-166.50,-6.00),v60,z5,tcp\WObj:=Plywood;
    MoveL Offs(pOrigin,130.10,-166.50,-6.00),vTravel,z5,tcp\WObj:=Plywood;
    MoveL Offs(pOrigin,130.10,-166.50,-0.00),v60,z0,tcp\WObj:=Plywood;
    MoveL Offs(pOrigin,129.36,-164.87,-0.00),v40,z0,tcp\WObj:=Plywood;
    MoveL Offs(pOrigin,129.68,-166.39,-0.00),v40,z0,tcp\WObj:=Plywood;
    MoveL Offs(pOrigin,129.46,-168.77,-0.00),v40,z0,tcp\WObj:=Plywood;
    MoveL Offs(pOrigin,129.99,-167.88,-0.00),v40,z0,tcp\WObj:=Plywood;
  ENDPROC

  PROC DrawPart20()
    MoveL Offs(pOrigin,130.10,-166.50,-0.00),v40,z0,tcp\WObj:=Plywood;
    MoveL Offs(pOrigin,129.14,-165.97,-0.00),v40,z0,tcp\WObj:=Plywood;
    MoveL Offs(pOrigin,128.75,-164.91,-0.00),v40,z0,tcp\WObj:=Plywood;
    MoveL Offs(pOrigin,127.76,-163.74,-0.00),v40,z0,tcp\WObj:=Plywood;
    MoveL Offs(pOrigin,127.30,-163.63,-0.00),v40,z0,tcp\WObj:=Plywood;
    MoveL Offs(pOrigin,128.29,-165.54,-0.00),v40,z0,tcp\WObj:=Plywood;
    MoveL Offs(pOrigin,128.19,-167.03,-0.00),v40,z0,tcp\WObj:=Plywood;
    MoveL Offs(pOrigin,127.80,-168.09,-0.00),v40,z0,tcp\WObj:=Plywood;
    MoveL Offs(pOrigin,126.77,-169.33,-0.00),v40,z0,tcp\WObj:=Plywood;
    MoveL Offs(pOrigin,127.76,-167.67,-0.00),v40,z0,tcp\WObj:=Plywood;
    MoveL Offs(pOrigin,127.62,-165.23,-0.00),v40,z0,tcp\WObj:=Plywood;
    MoveL Offs(pOrigin,126.06,-163.42,-0.00),v40,z0,tcp\WObj:=Plywood;
    MoveL Offs(pOrigin,123.44,-161.93,-0.00),v40,z0,tcp\WObj:=Plywood;
    MoveL Offs(pOrigin,126.31,-164.48,-0.00),v40,z0,tcp\WObj:=Plywood;
    MoveL Offs(pOrigin,126.91,-166.50,-0.00),v40,z0,tcp\WObj:=Plywood;
    MoveL Offs(pOrigin,126.70,-167.46,-0.00),v40,z0,tcp\WObj:=Plywood;
    MoveL Offs(pOrigin,125.43,-169.48,-0.00),v40,z0,tcp\WObj:=Plywood;
    MoveL Offs(pOrigin,123.41,-170.79,-0.00),v40,z0,tcp\WObj:=Plywood;
    MoveL Offs(pOrigin,121.18,-171.67,-0.00),v40,z0,tcp\WObj:=Plywood;
    MoveL Offs(pOrigin,121.07,-171.99,-0.00),v40,z0,tcp\WObj:=Plywood;
    MoveL Offs(pOrigin,124.04,-171.71,-0.00),v40,z0,tcp\WObj:=Plywood;
    MoveL Offs(pOrigin,126.17,-170.79,-0.00),v40,z0,tcp\WObj:=Plywood;
    MoveL Offs(pOrigin,127.87,-169.37,-0.00),v40,z0,tcp\WObj:=Plywood;
    MoveL Offs(pOrigin,128.44,-168.48,-0.00),v40,z0,tcp\WObj:=Plywood;
    MoveL Offs(pOrigin,127.27,-170.64,-0.00),v40,z0,tcp\WObj:=Plywood;
    MoveL Offs(pOrigin,127.97,-170.32,-0.00),v40,z0,tcp\WObj:=Plywood;
    MoveL Offs(pOrigin,128.93,-168.62,-0.00),v40,z0,tcp\WObj:=Plywood;
    MoveL Offs(pOrigin,129.14,-165.97,-0.00),v40,fine,tcp\WObj:=Plywood;
    MoveL Offs(pOrigin,129.14,-165.97,-6.00),v60,z5,tcp\WObj:=Plywood;
    MoveL Offs(pOrigin,126.38,-166.93,-6.00),vTravel,z5,tcp\WObj:=Plywood;
    MoveL Offs(pOrigin,126.38,-166.93,-0.00),v60,z0,tcp\WObj:=Plywood;
    MoveL Offs(pOrigin,126.20,-165.44,-0.00),v40,z0,tcp\WObj:=Plywood;
    MoveL Offs(pOrigin,125.43,-164.16,-0.00),v40,z0,tcp\WObj:=Plywood;
    MoveL Offs(pOrigin,125.60,-165.15,-0.00),v40,z0,tcp\WObj:=Plywood;
    MoveL Offs(pOrigin,124.47,-163.63,-0.00),v40,z0,tcp\WObj:=Plywood;
    MoveL Offs(pOrigin,121.92,-161.93,-0.00),v40,z0,tcp\WObj:=Plywood;
    MoveL Offs(pOrigin,121.18,-161.05,-0.00),v40,z0,tcp\WObj:=Plywood;
    MoveL Offs(pOrigin,121.60,-162.14,-0.00),v40,z0,tcp\WObj:=Plywood;
    MoveL Offs(pOrigin,123.62,-163.52,-0.00),v40,z0,tcp\WObj:=Plywood;
    MoveL Offs(pOrigin,125.14,-165.54,-0.00),v40,z0,tcp\WObj:=Plywood;
    MoveL Offs(pOrigin,125.43,-167.56,-0.00),v40,z0,tcp\WObj:=Plywood;
    MoveL Offs(pOrigin,124.57,-169.65,-0.00),v40,z0,tcp\WObj:=Plywood;
    MoveL Offs(pOrigin,126.10,-167.77,-0.00),v40,z0,tcp\WObj:=Plywood;
    MoveL Offs(pOrigin,126.38,-166.93,-0.00),v40,fine,tcp\WObj:=Plywood;
    MoveL Offs(pOrigin,126.38,-166.93,-6.00),v60,z5,tcp\WObj:=Plywood;
    MoveL Offs(pOrigin,125.04,-167.35,-6.00),vTravel,z5,tcp\WObj:=Plywood;
    MoveL Offs(pOrigin,125.04,-167.35,-0.00),v60,z0,tcp\WObj:=Plywood;
    MoveL Offs(pOrigin,124.79,-165.86,-0.00),v40,z0,tcp\WObj:=Plywood;
    MoveL Offs(pOrigin,124.15,-164.59,-0.00),v40,z0,tcp\WObj:=Plywood;
    MoveL Offs(pOrigin,123.87,-164.48,-0.00),v40,z0,tcp\WObj:=Plywood;
    MoveL Offs(pOrigin,123.94,-164.84,-0.00),v40,z0,tcp\WObj:=Plywood;
    MoveL Offs(pOrigin,122.77,-163.63,-0.00),v40,z0,tcp\WObj:=Plywood;
    MoveL Offs(pOrigin,121.32,-162.78,-0.00),v40,z0,tcp\WObj:=Plywood;
    MoveL Offs(pOrigin,123.09,-164.69,-0.00),v40,z0,tcp\WObj:=Plywood;
    MoveL Offs(pOrigin,123.72,-166.18,-0.00),v40,z0,tcp\WObj:=Plywood;
    MoveL Offs(pOrigin,123.83,-167.46,-0.00),v40,z0,tcp\WObj:=Plywood;
    MoveL Offs(pOrigin,123.23,-169.05,-0.00),v40,z0,tcp\WObj:=Plywood;
    MoveL Offs(pOrigin,122.24,-170.11,-0.00),v40,z0,tcp\WObj:=Plywood;
    MoveL Offs(pOrigin,120.54,-171.10,-0.00),v40,z0,tcp\WObj:=Plywood;
    MoveL Offs(pOrigin,116.07,-172.10,-0.00),v40,z0,tcp\WObj:=Plywood;
    MoveL Offs(pOrigin,118.20,-172.13,-0.00),v40,z0,tcp\WObj:=Plywood;
    MoveL Offs(pOrigin,119.90,-171.71,-0.00),v40,z0,tcp\WObj:=Plywood;
    MoveL Offs(pOrigin,122.56,-170.57,-0.00),v40,z0,tcp\WObj:=Plywood;
    MoveL Offs(pOrigin,123.94,-169.58,-0.00),v40,z0,tcp\WObj:=Plywood;
    MoveL Offs(pOrigin,124.82,-168.31,-0.00),v40,z0,tcp\WObj:=Plywood;
    MoveL Offs(pOrigin,125.04,-167.35,-0.00),v40,fine,tcp\WObj:=Plywood;
    MoveL Offs(pOrigin,125.04,-167.35,-6.00),v60,z5,tcp\WObj:=Plywood;
    MoveL Offs(pOrigin,123.48,-167.03,-6.00),vTravel,z5,tcp\WObj:=Plywood;
    MoveL Offs(pOrigin,123.48,-167.03,-0.00),v60,z0,tcp\WObj:=Plywood;
    MoveL Offs(pOrigin,122.77,-165.23,-0.00),v40,z0,tcp\WObj:=Plywood;
    MoveL Offs(pOrigin,121.39,-164.13,-0.00),v40,z0,tcp\WObj:=Plywood;
    MoveL Offs(pOrigin,122.20,-165.33,-0.00),v40,z0,tcp\WObj:=Plywood;
    MoveL Offs(pOrigin,122.66,-166.93,-0.00),v40,z0,tcp\WObj:=Plywood;
    MoveL Offs(pOrigin,122.56,-168.20,-0.00),v40,z0,tcp\WObj:=Plywood;
    MoveL Offs(pOrigin,121.71,-170.11,-0.00),v40,z0,tcp\WObj:=Plywood;
    MoveL Offs(pOrigin,123.12,-168.52,-0.00),v40,z0,tcp\WObj:=Plywood;
    MoveL Offs(pOrigin,123.48,-167.03,-0.00),v40,fine,tcp\WObj:=Plywood;
    MoveL Offs(pOrigin,123.48,-167.03,-6.00),v60,z5,tcp\WObj:=Plywood;
    MoveL Offs(pOrigin,120.43,-166.82,-6.00),vTravel,z5,tcp\WObj:=Plywood;
    MoveL Offs(pOrigin,120.43,-166.82,-0.00),v60,z0,tcp\WObj:=Plywood;
    MoveL Offs(pOrigin,120.01,-165.72,-0.00),v40,z0,tcp\WObj:=Plywood;
    MoveL Offs(pOrigin,119.90,-167.88,-0.00),v40,z0,tcp\WObj:=Plywood;
    MoveL Offs(pOrigin,118.94,-169.44,-0.00),v40,z0,tcp\WObj:=Plywood;
    MoveL Offs(pOrigin,119.90,-168.73,-0.00),v40,z0,tcp\WObj:=Plywood;
    MoveL Offs(pOrigin,120.32,-167.88,-0.00),v40,z0,tcp\WObj:=Plywood;
    MoveL Offs(pOrigin,120.43,-166.82,-0.00),v40,z0,tcp\WObj:=Plywood;
    MoveL Offs(pOrigin,119.79,-167.35,-0.00),v40,z0,tcp\WObj:=Plywood;
    MoveL Offs(pOrigin,119.19,-165.12,-0.00),v40,z0,tcp\WObj:=Plywood;
    MoveL Offs(pOrigin,117.67,-163.49,-0.00),v40,z0,tcp\WObj:=Plywood;
    MoveL Offs(pOrigin,117.49,-163.63,-0.00),v40,z0,tcp\WObj:=Plywood;
    MoveL Offs(pOrigin,118.77,-165.54,-0.00),v40,z0,tcp\WObj:=Plywood;
    MoveL Offs(pOrigin,118.94,-167.14,-0.00),v40,z0,tcp\WObj:=Plywood;
    MoveL Offs(pOrigin,118.09,-168.84,-0.00),v40,z0,tcp\WObj:=Plywood;
    MoveL Offs(pOrigin,116.71,-170.01,-0.00),v40,z0,tcp\WObj:=Plywood;
    MoveL Offs(pOrigin,118.94,-168.84,-0.00),v40,z0,tcp\WObj:=Plywood;
    MoveL Offs(pOrigin,119.79,-167.35,-0.00),v40,fine,tcp\WObj:=Plywood;
    MoveL Offs(pOrigin,119.79,-167.35,-6.00),v60,z5,tcp\WObj:=Plywood;
    MoveL Offs(pOrigin,118.27,-167.99,-6.00),vTravel,z5,tcp\WObj:=Plywood;
    MoveL Offs(pOrigin,118.27,-167.99,-0.00),v60,z0,tcp\WObj:=Plywood;
    MoveL Offs(pOrigin,118.52,-166.29,-0.00),v40,z0,tcp\WObj:=Plywood;
    MoveL Offs(pOrigin,118.24,-165.44,-0.00),v40,z0,tcp\WObj:=Plywood;
    MoveL Offs(pOrigin,115.76,-162.78,-0.00),v40,z0,tcp\WObj:=Plywood;
    MoveL Offs(pOrigin,115.61,-162.99,-0.00),v40,z0,tcp\WObj:=Plywood;
    MoveL Offs(pOrigin,116.64,-164.38,-0.00),v40,z0,tcp\WObj:=Plywood;
    MoveL Offs(pOrigin,117.03,-165.65,-0.00),v40,z0,tcp\WObj:=Plywood;
    MoveL Offs(pOrigin,116.64,-167.35,-0.00),v40,z0,tcp\WObj:=Plywood;
    MoveL Offs(pOrigin,115.44,-168.55,-0.00),v40,z0,tcp\WObj:=Plywood;
    MoveL Offs(pOrigin,111.61,-169.97,-0.00),v40,z0,tcp\WObj:=Plywood;
    MoveL Offs(pOrigin,115.76,-169.79,-0.00),v40,z0,tcp\WObj:=Plywood;
    MoveL Offs(pOrigin,117.24,-169.05,-0.00),v40,z0,tcp\WObj:=Plywood;
    MoveL Offs(pOrigin,118.27,-167.99,-0.00),v40,fine,tcp\WObj:=Plywood;
    MoveL Offs(pOrigin,118.27,-167.99,-6.00),v60,z5,tcp\WObj:=Plywood;
    MoveL Offs(pOrigin,116.61,-166.39,-6.00),vTravel,z5,tcp\WObj:=Plywood;
    MoveL Offs(pOrigin,116.61,-166.39,-0.00),v60,z0,tcp\WObj:=Plywood;
    MoveL Offs(pOrigin,116.22,-164.59,-0.00),v40,z0,tcp\WObj:=Plywood;
    MoveL Offs(pOrigin,114.91,-163.03,-0.00),v40,z0,tcp\WObj:=Plywood;
    MoveL Offs(pOrigin,115.54,-164.80,-0.00),v40,z0,tcp\WObj:=Plywood;
    MoveL Offs(pOrigin,115.54,-166.29,-0.00),v40,z0,tcp\WObj:=Plywood;
    MoveL Offs(pOrigin,114.06,-168.52,-0.00),v40,z0,tcp\WObj:=Plywood;
    MoveL Offs(pOrigin,115.76,-167.77,-0.00),v40,z0,tcp\WObj:=Plywood;
  ENDPROC

  PROC DrawPart21()
    MoveL Offs(pOrigin,116.61,-166.39,-0.00),v40,fine,tcp\WObj:=Plywood;
    MoveL Offs(pOrigin,116.61,-166.39,-6.00),v60,z5,tcp\WObj:=Plywood;
    MoveL Offs(pOrigin,115.12,-165.97,-6.00),vTravel,z5,tcp\WObj:=Plywood;
    MoveL Offs(pOrigin,115.12,-165.97,-0.00),v60,z0,tcp\WObj:=Plywood;
    MoveL Offs(pOrigin,114.94,-164.48,-0.00),v40,z0,tcp\WObj:=Plywood;
    MoveL Offs(pOrigin,112.78,-160.69,-0.00),v40,z0,tcp\WObj:=Plywood;
    MoveL Offs(pOrigin,112.85,-161.93,-0.00),v40,z0,tcp\WObj:=Plywood;
    MoveL Offs(pOrigin,114.16,-164.27,-0.00),v40,z0,tcp\WObj:=Plywood;
    MoveL Offs(pOrigin,114.16,-165.54,-0.00),v40,z0,tcp\WObj:=Plywood;
    MoveL Offs(pOrigin,113.21,-166.93,-0.00),v40,z0,tcp\WObj:=Plywood;
    MoveL Offs(pOrigin,111.29,-167.81,-0.00),v40,z0,tcp\WObj:=Plywood;
    MoveL Offs(pOrigin,111.40,-168.09,-0.00),v40,z0,tcp\WObj:=Plywood;
    MoveL Offs(pOrigin,112.57,-168.09,-0.00),v40,z0,tcp\WObj:=Plywood;
    MoveL Offs(pOrigin,113.95,-167.60,-0.00),v40,z0,tcp\WObj:=Plywood;
    MoveL Offs(pOrigin,114.69,-167.03,-0.00),v40,z0,tcp\WObj:=Plywood;
    MoveL Offs(pOrigin,115.12,-165.97,-0.00),v40,fine,tcp\WObj:=Plywood;
    MoveL Offs(pOrigin,115.12,-165.97,-6.00),v60,z5,tcp\WObj:=Plywood;
    MoveL Offs(pOrigin,113.95,-165.12,-6.00),vTravel,z5,tcp\WObj:=Plywood;
    MoveL Offs(pOrigin,113.95,-165.12,-0.00),v60,z0,tcp\WObj:=Plywood;
    MoveL Offs(pOrigin,113.35,-163.52,-0.00),v40,z0,tcp\WObj:=Plywood;
    MoveL Offs(pOrigin,112.14,-162.11,-0.00),v40,z0,tcp\WObj:=Plywood;
    MoveL Offs(pOrigin,112.99,-164.48,-0.00),v40,z0,tcp\WObj:=Plywood;
    MoveL Offs(pOrigin,112.99,-165.44,-0.00),v40,z0,tcp\WObj:=Plywood;
    MoveL Offs(pOrigin,112.07,-167.03,-0.00),v40,z0,tcp\WObj:=Plywood;
    MoveL Offs(pOrigin,112.25,-167.17,-0.00),v40,z0,tcp\WObj:=Plywood;
    MoveL Offs(pOrigin,113.63,-166.18,-0.00),v40,z0,tcp\WObj:=Plywood;
    MoveL Offs(pOrigin,113.95,-165.12,-0.00),v40,fine,tcp\WObj:=Plywood;
    MoveL Offs(pOrigin,113.95,-165.12,-6.00),v60,z5,tcp\WObj:=Plywood;
    MoveL Offs(pOrigin,112.68,-164.80,-6.00),vTravel,z5,tcp\WObj:=Plywood;
    MoveL Offs(pOrigin,112.68,-164.80,-0.00),v60,z0,tcp\WObj:=Plywood;
    MoveL Offs(pOrigin,111.86,-162.68,-0.00),v40,z0,tcp\WObj:=Plywood;
    MoveL Offs(pOrigin,110.76,-161.26,-0.00),v40,z0,tcp\WObj:=Plywood;
    MoveL Offs(pOrigin,111.93,-164.16,-0.00),v40,z0,tcp\WObj:=Plywood;
    MoveL Offs(pOrigin,111.65,-165.44,-0.00),v40,z0,tcp\WObj:=Plywood;
    MoveL Offs(pOrigin,110.87,-166.32,-0.00),v40,z0,tcp\WObj:=Plywood;
    MoveL Offs(pOrigin,109.06,-167.03,-0.00),v40,z0,tcp\WObj:=Plywood;
    MoveL Offs(pOrigin,106.94,-167.14,-0.00),v40,z0,tcp\WObj:=Plywood;
    MoveL Offs(pOrigin,103.36,-165.97,-0.00),v40,z0,tcp\WObj:=Plywood;
    MoveL Offs(pOrigin,104.28,-166.75,-0.00),v40,z0,tcp\WObj:=Plywood;
    MoveL Offs(pOrigin,107.47,-167.88,-0.00),v40,z0,tcp\WObj:=Plywood;
    MoveL Offs(pOrigin,109.49,-167.88,-0.00),v40,z0,tcp\WObj:=Plywood;
    MoveL Offs(pOrigin,111.82,-166.93,-0.00),v40,z0,tcp\WObj:=Plywood;
    MoveL Offs(pOrigin,112.60,-165.86,-0.00),v40,z0,tcp\WObj:=Plywood;
    MoveL Offs(pOrigin,112.68,-164.80,-0.00),v40,z0,tcp\WObj:=Plywood;
    MoveL Offs(pOrigin,111.61,-164.38,-0.00),v40,z0,tcp\WObj:=Plywood;
    MoveL Offs(pOrigin,111.33,-163.10,-0.00),v40,z0,tcp\WObj:=Plywood;
    MoveL Offs(pOrigin,111.01,-162.99,-0.00),v40,z0,tcp\WObj:=Plywood;
    MoveL Offs(pOrigin,111.19,-164.09,-0.00),v40,z0,tcp\WObj:=Plywood;
    MoveL Offs(pOrigin,110.34,-162.32,-0.00),v40,z0,tcp\WObj:=Plywood;
    MoveL Offs(pOrigin,110.44,-164.80,-0.00),v40,z0,tcp\WObj:=Plywood;
    MoveL Offs(pOrigin,109.17,-166.61,-0.00),v40,z0,tcp\WObj:=Plywood;
    MoveL Offs(pOrigin,110.76,-165.86,-0.00),v40,z0,tcp\WObj:=Plywood;
    MoveL Offs(pOrigin,111.61,-164.38,-0.00),v40,fine,tcp\WObj:=Plywood;
    MoveL Offs(pOrigin,111.61,-164.38,-6.00),v60,z5,tcp\WObj:=Plywood;
    MoveL Offs(pOrigin,110.34,-163.63,-6.00),vTravel,z5,tcp\WObj:=Plywood;
    MoveL Offs(pOrigin,110.34,-163.63,-0.00),v60,z0,tcp\WObj:=Plywood;
    MoveL Offs(pOrigin,109.49,-161.36,-0.00),v40,z0,tcp\WObj:=Plywood;
    MoveL Offs(pOrigin,109.42,-164.91,-0.00),v40,z0,tcp\WObj:=Plywood;
    MoveL Offs(pOrigin,107.36,-166.46,-0.00),v40,z0,tcp\WObj:=Plywood;
    MoveL Offs(pOrigin,109.06,-166.11,-0.00),v40,z0,tcp\WObj:=Plywood;
    MoveL Offs(pOrigin,110.16,-164.91,-0.00),v40,z0,tcp\WObj:=Plywood;
    MoveL Offs(pOrigin,110.34,-163.63,-0.00),v40,z0,tcp\WObj:=Plywood;
    MoveL Offs(pOrigin,109.38,-163.10,-0.00),v40,z0,tcp\WObj:=Plywood;
    MoveL Offs(pOrigin,108.85,-160.20,-0.00),v40,z0,tcp\WObj:=Plywood;
    MoveL Offs(pOrigin,108.53,-161.08,-0.00),v40,z0,tcp\WObj:=Plywood;
    MoveL Offs(pOrigin,108.64,-162.50,-0.00),v40,z0,tcp\WObj:=Plywood;
    MoveL Offs(pOrigin,108.43,-161.51,-0.00),v40,z0,tcp\WObj:=Plywood;
    MoveL Offs(pOrigin,108.71,-159.27,-0.00),v40,z0,tcp\WObj:=Plywood;
    MoveL Offs(pOrigin,107.86,-160.66,-0.00),v40,z0,tcp\WObj:=Plywood;
    MoveL Offs(pOrigin,107.68,-162.68,-0.00),v40,z0,tcp\WObj:=Plywood;
    MoveL Offs(pOrigin,107.15,-163.95,-0.00),v40,z0,tcp\WObj:=Plywood;
    MoveL Offs(pOrigin,105.03,-164.91,-0.00),v40,z0,tcp\WObj:=Plywood;
    MoveL Offs(pOrigin,103.43,-165.01,-0.00),v40,z0,tcp\WObj:=Plywood;
    MoveL Offs(pOrigin,104.71,-165.44,-0.00),v40,z0,tcp\WObj:=Plywood;
    MoveL Offs(pOrigin,106.41,-165.44,-0.00),v40,z0,tcp\WObj:=Plywood;
    MoveL Offs(pOrigin,107.61,-164.94,-0.00),v40,z0,tcp\WObj:=Plywood;
    MoveL Offs(pOrigin,106.30,-165.65,-0.00),v40,z0,tcp\WObj:=Plywood;
    MoveL Offs(pOrigin,104.78,-165.65,-0.00),v40,z0,tcp\WObj:=Plywood;
    MoveL Offs(pOrigin,105.77,-166.07,-0.00),v40,z0,tcp\WObj:=Plywood;
    MoveL Offs(pOrigin,107.26,-166.07,-0.00),v40,z0,tcp\WObj:=Plywood;
    MoveL Offs(pOrigin,109.28,-164.91,-0.00),v40,z0,tcp\WObj:=Plywood;
    MoveL Offs(pOrigin,109.38,-163.10,-0.00),v40,fine,tcp\WObj:=Plywood;
    MoveL Offs(pOrigin,109.38,-163.10,-6.00),v60,z5,tcp\WObj:=Plywood;
    MoveL Offs(pOrigin,110.02,-161.58,-6.00),vTravel,z5,tcp\WObj:=Plywood;
    MoveL Offs(pOrigin,110.02,-161.58,-0.00),v60,z0,tcp\WObj:=Plywood;
    MoveL Offs(pOrigin,110.34,-159.35,-0.00),v40,z0,tcp\WObj:=Plywood;
    MoveL Offs(pOrigin,109.81,-160.55,-0.00),v40,z0,tcp\WObj:=Plywood;
    MoveL Offs(pOrigin,110.02,-161.58,-0.00),v40,fine,tcp\WObj:=Plywood;
    MoveL Offs(pOrigin,110.02,-161.58,-6.00),v60,z5,tcp\WObj:=Plywood;
    MoveL Offs(pOrigin,107.57,-162.57,-6.00),vTravel,z5,tcp\WObj:=Plywood;
    MoveL Offs(pOrigin,107.57,-162.57,-0.00),v60,z0,tcp\WObj:=Plywood;
    MoveL Offs(pOrigin,107.75,-159.91,-0.00),v40,z0,tcp\WObj:=Plywood;
    MoveL Offs(pOrigin,108.85,-158.14,-0.00),v40,z0,tcp\WObj:=Plywood;
    MoveL Offs(pOrigin,107.33,-159.59,-0.00),v40,z0,tcp\WObj:=Plywood;
    MoveL Offs(pOrigin,106.19,-163.17,-0.00),v40,z0,tcp\WObj:=Plywood;
    MoveL Offs(pOrigin,105.98,-162.60,-0.00),v40,z0,tcp\WObj:=Plywood;
    MoveL Offs(pOrigin,104.07,-163.84,-0.00),v40,z0,tcp\WObj:=Plywood;
    MoveL Offs(pOrigin,100.99,-163.42,-0.00),v40,z0,tcp\WObj:=Plywood;
    MoveL Offs(pOrigin,102.16,-164.09,-0.00),v40,z0,tcp\WObj:=Plywood;
    MoveL Offs(pOrigin,104.18,-164.59,-0.00),v40,z0,tcp\WObj:=Plywood;
    MoveL Offs(pOrigin,105.34,-164.48,-0.00),v40,z0,tcp\WObj:=Plywood;
    MoveL Offs(pOrigin,106.41,-163.91,-0.00),v40,z0,tcp\WObj:=Plywood;
    MoveL Offs(pOrigin,106.83,-164.06,-0.00),v40,z0,tcp\WObj:=Plywood;
    MoveL Offs(pOrigin,107.57,-162.57,-0.00),v40,fine,tcp\WObj:=Plywood;
    MoveL Offs(pOrigin,107.57,-162.57,-6.00),v60,z5,tcp\WObj:=Plywood;
    MoveL Offs(pOrigin,106.16,-161.82,-6.00),vTravel,z5,tcp\WObj:=Plywood;
    MoveL Offs(pOrigin,106.16,-161.82,-0.00),v60,z0,tcp\WObj:=Plywood;
    MoveL Offs(pOrigin,105.98,-161.65,-0.00),v40,z0,tcp\WObj:=Plywood;
    MoveL Offs(pOrigin,104.39,-162.68,-0.00),v40,z0,tcp\WObj:=Plywood;
    MoveL Offs(pOrigin,102.58,-162.89,-0.00),v40,z0,tcp\WObj:=Plywood;
    MoveL Offs(pOrigin,100.24,-161.72,-0.00),v40,z0,tcp\WObj:=Plywood;
    MoveL Offs(pOrigin,97.94,-159.70,-0.00),v40,z0,tcp\WObj:=Plywood;
    MoveL Offs(pOrigin,98.97,-161.47,-0.00),v40,z0,tcp\WObj:=Plywood;
    MoveL Offs(pOrigin,100.78,-162.82,-0.00),v40,z0,tcp\WObj:=Plywood;
    MoveL Offs(pOrigin,101.84,-163.21,-0.00),v40,z0,tcp\WObj:=Plywood;
    MoveL Offs(pOrigin,104.07,-163.31,-0.00),v40,z0,tcp\WObj:=Plywood;
    MoveL Offs(pOrigin,105.24,-162.78,-0.00),v40,z0,tcp\WObj:=Plywood;
    MoveL Offs(pOrigin,106.16,-161.82,-0.00),v40,z0,tcp\WObj:=Plywood;
    MoveL Offs(pOrigin,106.02,-161.19,-0.00),v40,z0,tcp\WObj:=Plywood;
    MoveL Offs(pOrigin,107.01,-158.21,-0.00),v40,z0,tcp\WObj:=Plywood;
  ENDPROC

  PROC DrawPart22()
    MoveL Offs(pOrigin,105.34,-159.98,-0.00),v40,z0,tcp\WObj:=Plywood;
    MoveL Offs(pOrigin,102.83,-160.98,-0.00),v40,z0,tcp\WObj:=Plywood;
    MoveL Offs(pOrigin,103.86,-161.08,-0.00),v40,z0,tcp\WObj:=Plywood;
    MoveL Offs(pOrigin,105.91,-160.27,-0.00),v40,z0,tcp\WObj:=Plywood;
    MoveL Offs(pOrigin,104.39,-161.22,-0.00),v40,z0,tcp\WObj:=Plywood;
    MoveL Offs(pOrigin,102.26,-161.51,-0.00),v40,z0,tcp\WObj:=Plywood;
    MoveL Offs(pOrigin,100.10,-161.08,-0.00),v40,z0,tcp\WObj:=Plywood;
    MoveL Offs(pOrigin,102.37,-162.46,-0.00),v40,z0,tcp\WObj:=Plywood;
    MoveL Offs(pOrigin,104.49,-162.39,-0.00),v40,z0,tcp\WObj:=Plywood;
    MoveL Offs(pOrigin,106.02,-161.19,-0.00),v40,fine,tcp\WObj:=Plywood;
    MoveL Offs(pOrigin,106.02,-161.19,-6.00),v60,z5,tcp\WObj:=Plywood;
    MoveL Offs(pOrigin,103.96,-160.27,-6.00),vTravel,z5,tcp\WObj:=Plywood;
    MoveL Offs(pOrigin,103.96,-160.27,-0.00),v60,z0,tcp\WObj:=Plywood;
    MoveL Offs(pOrigin,107.72,-157.26,-0.00),v40,z0,tcp\WObj:=Plywood;
    MoveL Offs(pOrigin,105.88,-157.86,-0.00),v40,z0,tcp\WObj:=Plywood;
    MoveL Offs(pOrigin,102.58,-159.84,-0.00),v40,z0,tcp\WObj:=Plywood;
    MoveL Offs(pOrigin,99.85,-159.91,-0.00),v40,z0,tcp\WObj:=Plywood;
    MoveL Offs(pOrigin,101.31,-160.55,-0.00),v40,z0,tcp\WObj:=Plywood;
    MoveL Offs(pOrigin,103.96,-160.27,-0.00),v40,z0,tcp\WObj:=Plywood;
    MoveL Offs(pOrigin,103.32,-159.31,-0.00),v40,z0,tcp\WObj:=Plywood;
    MoveL Offs(pOrigin,106.69,-156.62,-0.00),v40,z0,tcp\WObj:=Plywood;
    MoveL Offs(pOrigin,101.94,-158.64,-0.00),v40,z0,tcp\WObj:=Plywood;
    MoveL Offs(pOrigin,100.03,-158.64,-0.00),v40,z0,tcp\WObj:=Plywood;
    MoveL Offs(pOrigin,98.86,-158.25,-0.00),v40,z0,tcp\WObj:=Plywood;
    MoveL Offs(pOrigin,97.27,-156.73,-0.00),v40,z0,tcp\WObj:=Plywood;
    MoveL Offs(pOrigin,97.06,-156.83,-0.00),v40,z0,tcp\WObj:=Plywood;
    MoveL Offs(pOrigin,98.97,-159.10,-0.00),v40,z0,tcp\WObj:=Plywood;
    MoveL Offs(pOrigin,101.62,-159.81,-0.00),v40,z0,tcp\WObj:=Plywood;
    MoveL Offs(pOrigin,103.32,-159.31,-0.00),v40,fine,tcp\WObj:=Plywood;
    MoveL Offs(pOrigin,103.32,-159.31,-6.00),v60,z5,tcp\WObj:=Plywood;
    MoveL Offs(pOrigin,102.58,-158.11,-6.00),vTravel,z5,tcp\WObj:=Plywood;
    MoveL Offs(pOrigin,102.58,-158.11,-0.00),v60,z0,tcp\WObj:=Plywood;
    MoveL Offs(pOrigin,104.60,-156.83,-0.00),v40,z0,tcp\WObj:=Plywood;
    MoveL Offs(pOrigin,104.49,-156.62,-0.00),v40,z0,tcp\WObj:=Plywood;
    MoveL Offs(pOrigin,103.11,-157.43,-0.00),v40,z0,tcp\WObj:=Plywood;
    MoveL Offs(pOrigin,101.84,-157.68,-0.00),v40,z0,tcp\WObj:=Plywood;
    MoveL Offs(pOrigin,103.36,-157.04,-0.00),v40,z0,tcp\WObj:=Plywood;
    MoveL Offs(pOrigin,99.18,-156.23,-0.00),v40,z0,tcp\WObj:=Plywood;
    MoveL Offs(pOrigin,96.24,-153.96,-0.00),v40,z0,tcp\WObj:=Plywood;
    MoveL Offs(pOrigin,96.60,-155.02,-0.00),v40,z0,tcp\WObj:=Plywood;
    MoveL Offs(pOrigin,98.37,-156.90,-0.00),v40,z0,tcp\WObj:=Plywood;
    MoveL Offs(pOrigin,98.22,-157.15,-0.00),v40,z0,tcp\WObj:=Plywood;
    MoveL Offs(pOrigin,99.71,-158.04,-0.00),v40,z0,tcp\WObj:=Plywood;
    MoveL Offs(pOrigin,100.78,-158.32,-0.00),v40,z0,tcp\WObj:=Plywood;
    MoveL Offs(pOrigin,102.58,-158.11,-0.00),v40,fine,tcp\WObj:=Plywood;
    MoveL Offs(pOrigin,102.58,-158.11,-6.00),v60,z5,tcp\WObj:=Plywood;
    MoveL Offs(pOrigin,103.01,-156.62,-6.00),vTravel,z5,tcp\WObj:=Plywood;
    MoveL Offs(pOrigin,103.01,-156.62,-0.00),v60,z0,tcp\WObj:=Plywood;
    MoveL Offs(pOrigin,103.57,-156.30,-0.00),v40,z0,tcp\WObj:=Plywood;
    MoveL Offs(pOrigin,102.16,-156.41,-0.00),v40,z0,tcp\WObj:=Plywood;
    MoveL Offs(pOrigin,103.01,-156.62,-0.00),v40,fine,tcp\WObj:=Plywood;
    MoveL Offs(pOrigin,103.01,-156.62,-6.00),v60,z5,tcp\WObj:=Plywood;
    MoveL Offs(pOrigin,101.77,-156.09,-6.00),vTravel,z5,tcp\WObj:=Plywood;
    MoveL Offs(pOrigin,101.77,-156.09,-0.00),v60,z0,tcp\WObj:=Plywood;
    MoveL Offs(pOrigin,100.39,-155.38,-0.00),v40,z0,tcp\WObj:=Plywood;
    MoveL Offs(pOrigin,101.73,-155.77,-0.00),v40,z0,tcp\WObj:=Plywood;
    MoveL Offs(pOrigin,104.07,-155.63,-0.00),v40,z0,tcp\WObj:=Plywood;
    MoveL Offs(pOrigin,100.56,-154.74,-0.00),v40,z0,tcp\WObj:=Plywood;
    MoveL Offs(pOrigin,98.65,-153.64,-0.00),v40,z0,tcp\WObj:=Plywood;
    MoveL Offs(pOrigin,96.67,-150.46,-0.00),v40,z0,tcp\WObj:=Plywood;
    MoveL Offs(pOrigin,96.74,-151.73,-0.00),v40,z0,tcp\WObj:=Plywood;
    MoveL Offs(pOrigin,97.30,-153.22,-0.00),v40,z0,tcp\WObj:=Plywood;
    MoveL Offs(pOrigin,98.76,-155.02,-0.00),v40,z0,tcp\WObj:=Plywood;
    MoveL Offs(pOrigin,101.20,-156.19,-0.00),v40,z0,tcp\WObj:=Plywood;
    MoveL Offs(pOrigin,101.77,-156.09,-0.00),v40,fine,tcp\WObj:=Plywood;
    MoveL Offs(pOrigin,101.77,-156.09,-6.00),v60,z5,tcp\WObj:=Plywood;
    MoveL Offs(pOrigin,102.16,-154.81,-6.00),vTravel,z5,tcp\WObj:=Plywood;
    MoveL Offs(pOrigin,102.16,-154.81,-0.00),v60,z0,tcp\WObj:=Plywood;
    MoveL Offs(pOrigin,102.37,-154.60,-0.00),v40,z0,tcp\WObj:=Plywood;
    MoveL Offs(pOrigin,101.20,-154.10,-0.00),v40,z0,tcp\WObj:=Plywood;
    MoveL Offs(pOrigin,100.10,-153.15,-0.00),v40,z0,tcp\WObj:=Plywood;
    MoveL Offs(pOrigin,102.47,-154.18,-0.00),v40,z0,tcp\WObj:=Plywood;
    MoveL Offs(pOrigin,103.32,-154.14,-0.00),v40,z0,tcp\WObj:=Plywood;
    MoveL Offs(pOrigin,100.88,-153.04,-0.00),v40,z0,tcp\WObj:=Plywood;
    MoveL Offs(pOrigin,99.07,-151.70,-0.00),v40,z0,tcp\WObj:=Plywood;
    MoveL Offs(pOrigin,96.67,-148.54,-0.00),v40,z0,tcp\WObj:=Plywood;
    MoveL Offs(pOrigin,97.87,-151.73,-0.00),v40,z0,tcp\WObj:=Plywood;
    MoveL Offs(pOrigin,99.07,-153.32,-0.00),v40,z0,tcp\WObj:=Plywood;
    MoveL Offs(pOrigin,100.35,-154.21,-0.00),v40,z0,tcp\WObj:=Plywood;
    MoveL Offs(pOrigin,102.16,-154.81,-0.00),v40,fine,tcp\WObj:=Plywood;
    MoveL Offs(pOrigin,102.16,-154.81,-6.00),v60,z5,tcp\WObj:=Plywood;
    MoveL Offs(pOrigin,102.47,-153.08,-6.00),vTravel,z5,tcp\WObj:=Plywood;
    MoveL Offs(pOrigin,102.47,-153.08,-0.00),v60,z0,tcp\WObj:=Plywood;
    MoveL Offs(pOrigin,99.61,-150.46,-0.00),v40,z0,tcp\WObj:=Plywood;
    MoveL Offs(pOrigin,96.35,-146.21,-0.00),v40,z0,tcp\WObj:=Plywood;
    MoveL Offs(pOrigin,98.86,-150.99,-0.00),v40,z0,tcp\WObj:=Plywood;
    MoveL Offs(pOrigin,100.46,-152.30,-0.00),v40,z0,tcp\WObj:=Plywood;
    MoveL Offs(pOrigin,102.47,-153.08,-0.00),v40,z0,tcp\WObj:=Plywood;
    MoveL Offs(pOrigin,102.79,-152.55,-0.00),v40,z0,tcp\WObj:=Plywood;
    MoveL Offs(pOrigin,102.47,-152.05,-0.00),v40,z0,tcp\WObj:=Plywood;
    MoveL Offs(pOrigin,100.60,-150.99,-0.00),v40,z0,tcp\WObj:=Plywood;
    MoveL Offs(pOrigin,102.79,-152.55,-0.00),v40,fine,tcp\WObj:=Plywood;
    MoveL Offs(pOrigin,102.79,-152.55,-6.00),v60,z5,tcp\WObj:=Plywood;
    MoveL Offs(pOrigin,102.26,-150.42,-6.00),vTravel,z5,tcp\WObj:=Plywood;
    MoveL Offs(pOrigin,102.26,-150.42,-0.00),v60,z0,tcp\WObj:=Plywood;
    MoveL Offs(pOrigin,99.39,-146.10,-0.00),v40,z0,tcp\WObj:=Plywood;
    MoveL Offs(pOrigin,98.15,-144.93,-0.00),v40,z0,tcp\WObj:=Plywood;
    MoveL Offs(pOrigin,99.71,-147.80,-0.00),v40,z0,tcp\WObj:=Plywood;
    MoveL Offs(pOrigin,102.26,-150.42,-0.00),v40,z0,tcp\WObj:=Plywood;
    MoveL Offs(pOrigin,101.20,-150.85,-0.00),v40,z0,tcp\WObj:=Plywood;
    MoveL Offs(pOrigin,97.30,-144.82,-0.00),v40,z0,tcp\WObj:=Plywood;
    MoveL Offs(pOrigin,97.76,-147.06,-0.00),v40,z0,tcp\WObj:=Plywood;
    MoveL Offs(pOrigin,98.51,-148.33,-0.00),v40,z0,tcp\WObj:=Plywood;
    MoveL Offs(pOrigin,100.14,-150.24,-0.00),v40,z0,tcp\WObj:=Plywood;
    MoveL Offs(pOrigin,101.20,-150.85,-0.00),v40,fine,tcp\WObj:=Plywood;
    MoveL Offs(pOrigin,101.20,-150.85,-6.00),v60,z5,tcp\WObj:=Plywood;
    MoveL Offs(pOrigin,100.03,-148.86,-6.00),vTravel,z5,tcp\WObj:=Plywood;
    MoveL Offs(pOrigin,100.03,-148.86,-0.00),v60,z0,tcp\WObj:=Plywood;
    MoveL Offs(pOrigin,99.82,-148.33,-0.00),v40,z0,tcp\WObj:=Plywood;
    MoveL Offs(pOrigin,100.03,-148.86,-0.00),v40,fine,tcp\WObj:=Plywood;
    MoveL Offs(pOrigin,100.03,-148.86,-6.00),v60,z5,tcp\WObj:=Plywood;
    MoveL Offs(pOrigin,101.48,-148.33,-6.00),vTravel,z5,tcp\WObj:=Plywood;
    MoveL Offs(pOrigin,101.48,-148.33,-0.00),v60,z0,tcp\WObj:=Plywood;
    MoveL Offs(pOrigin,101.34,-147.27,-0.00),v40,z0,tcp\WObj:=Plywood;
    MoveL Offs(pOrigin,100.39,-145.46,-0.00),v40,z0,tcp\WObj:=Plywood;
    MoveL Offs(pOrigin,98.54,-143.48,-0.00),v40,z0,tcp\WObj:=Plywood;
    MoveL Offs(pOrigin,101.48,-148.33,-0.00),v40,fine,tcp\WObj:=Plywood;
    MoveL Offs(pOrigin,101.48,-148.33,-6.00),v60,z5,tcp\WObj:=Plywood;
    MoveL Offs(pOrigin,101.27,-145.36,-6.00),vTravel,z5,tcp\WObj:=Plywood;
    MoveL Offs(pOrigin,101.27,-145.36,-0.00),v60,z0,tcp\WObj:=Plywood;
  ENDPROC

